Omron Sysmac Studio project 17-701_20171123 (Sysmac Studio 1.19.0.13, StandardProject)

# Controller new_Controller_0: NJ101-1000 version 1.13
Units and slaves: 電源 : NJ-Px3001; CPU : NJ101-1000; 0 : CJ1W-ID211 (J01); 1 : CJ1W-OD211 (J02)
Task PrimaryTask (priority 4, period or condition 2000): prIndexDataChange, prIndex, prStation1_PanelLoad, prStation1_FeedPanelLoad, prError, prStation1_PanelUnLoad, prStation1_FeedPanelUnLoad, prSystemInit, prStation1, prStation16, prStation4, prStation4_TH, prStation2

TYPE stIndexData : STRUCT
    FinishFlag : ARRAY[0..19] OF BOOL;
    OKFlag : ARRAY[0..19] OF BOOL;
    NGFlag : ARRAY[0..19] OF BOOL;
    ErrorLog : ARRAY[0..19] OF INT;
END_STRUCT END_TYPE

VAR_GLOBAL
    LS_S1_Load_PanelUpDown1Back : BOOL;  (* at ECAT://node#[1,1]/Input Bit 16 bits/Input Bit 00; published *)
    LS_S1_Load_PanelUpDown1Out : BOOL;  (* at ECAT://node#[1,1]/Input Bit 16 bits/Input Bit 01; published *)
    LS_S1_Load_PanelUpDown2Back : BOOL;  (* at ECAT://node#[1,1]/Input Bit 16 bits/Input Bit 02; published *)
    LS_S1_Load_PanelUpDown2Out : BOOL;  (* at ECAT://node#[1,1]/Input Bit 16 bits/Input Bit 03; published *)
    LS_S1_Load_PanelClip1Back : BOOL;  (* at ECAT://node#[1,1]/Input Bit 16 bits/Input Bit 04; published *)
    LS_S1_Load_PanelClip1Out : BOOL;  (* at ECAT://node#[1,1]/Input Bit 16 bits/Input Bit 05; published *)
    LS_S1_Load_PanelClip2Back : BOOL;  (* at ECAT://node#[1,1]/Input Bit 16 bits/Input Bit 06; published *)
    LS_S1_Load_PanelClip2Out : BOOL;  (* at ECAT://node#[1,1]/Input Bit 16 bits/Input Bit 07; published *)
    LS_S1_Load_FixClipBack : BOOL;  (* at ECAT://node#[1,1]/Input Bit 16 bits/Input Bit 08; published *)
    LS_S1_Load_FixClipOut : BOOL;  (* at ECAT://node#[1,1]/Input Bit 16 bits/Input Bit 09; published *)
    LS_S1_Load_AlignmentClipBack : BOOL;  (* at ECAT://node#[1,1]/Input Bit 16 bits/Input Bit 10; published *)
    LS_S1_Load_AlignmentClipOut : BOOL;  (* at ECAT://node#[1,1]/Input Bit 16 bits/Input Bit 11; published *)
    LS_S1_Load_ConveyorClip1Back : BOOL;  (* at ECAT://node#[1,1]/Input Bit 16 bits/Input Bit 12; published *)
    LS_S1_Load_ConveyorClip1Out : BOOL;  (* at ECAT://node#[1,1]/Input Bit 16 bits/Input Bit 13; published *)
    LS_S1_Load_ConveyorClip2Back : BOOL;  (* at ECAT://node#[1,1]/Input Bit 16 bits/Input Bit 14; published *)
    LS_S1_Load_ConveyorClip2Out : BOOL;  (* at ECAT://node#[1,1]/Input Bit 16 bits/Input Bit 15; published *)
    LS_S1_Load_UpDownBack : BOOL;  (* at ECAT://node#[1,2]/Input Bit 16 bits/Input Bit 00; published *)
    LS_S1_Load_UpDownOut : BOOL;  (* at ECAT://node#[1,2]/Input Bit 16 bits/Input Bit 01; published *)
    LS_S1_UnLoad_UpDownBack : BOOL;  (* at ECAT://node#[1,2]/Input Bit 16 bits/Input Bit 02; published *)
    LS_S1_UnLoad_UpDownOut : BOOL;  (* at ECAT://node#[1,2]/Input Bit 16 bits/Input Bit 03; published *)
    LS_S1_UnLoad_ConveyorClip1Back : BOOL;  (* at ECAT://node#[1,2]/Input Bit 16 bits/Input Bit 04; published *)
    LS_S1_UnLoad_ConveyorClip1Out : BOOL;  (* at ECAT://node#[1,2]/Input Bit 16 bits/Input Bit 05; published *)
    LS_S1_UnLoad_ConveyorClip2Back : BOOL;  (* at ECAT://node#[1,2]/Input Bit 16 bits/Input Bit 06; published *)
    LS_S1_UnLoad_ConveyorClip2Out : BOOL;  (* at ECAT://node#[1,2]/Input Bit 16 bits/Input Bit 07; published *)
    LS_S1_UnLoad_FixClipBack : BOOL;  (* at ECAT://node#[1,2]/Input Bit 16 bits/Input Bit 08; published *)
    LS_S1_UnLoad_FixClipOut : BOOL;  (* at ECAT://node#[1,2]/Input Bit 16 bits/Input Bit 09; published *)
    LS_S1_UnLoad_AlignmentClipBack : BOOL;  (* at ECAT://node#[1,2]/Input Bit 16 bits/Input Bit 10; published *)
    LS_S1_UnLoad_AlignmentClipOut : BOOL;  (* at ECAT://node#[1,2]/Input Bit 16 bits/Input Bit 11; published *)
    LS_S1_UnLoad_PanelClip1Back : BOOL;  (* at ECAT://node#[1,2]/Input Bit 16 bits/Input Bit 12; published *)
    LS_S1_UnLoad_PanelClip1Out : BOOL;  (* at ECAT://node#[1,2]/Input Bit 16 bits/Input Bit 13; published *)
    LS_S1_UnLoad_PanelClip2Back : BOOL;  (* at ECAT://node#[1,2]/Input Bit 16 bits/Input Bit 14; published *)
    LS_S1_UnLoad_PanelClip2Out : BOOL;  (* at ECAT://node#[1,2]/Input Bit 16 bits/Input Bit 15; published *)
    LS_S1_UnLoad_PanelUpDown1Back : BOOL;  (* at ECAT://node#[1,3]/Input Bit 16 bits/Input Bit 00; published *)
    LS_S1_UnLoad_PanelUpDown1Out : BOOL;  (* at ECAT://node#[1,3]/Input Bit 16 bits/Input Bit 01; published *)
    LS_S1_UnLoad_PanelUpDown2Back : BOOL;  (* at ECAT://node#[1,3]/Input Bit 16 bits/Input Bit 02; published *)
    LS_S1_UnLoad_PanelUpDown2Out : BOOL;  (* at ECAT://node#[1,3]/Input Bit 16 bits/Input Bit 03; published *)
    SNR_S1_Load_Full : BOOL;  (* 出盤缺盤檢知; at ECAT://node#[1,3]/Input Bit 16 bits/Input Bit 08; published *)
    SNR_S1_UnLoad_Full : BOOL;  (* 收盤滿盤檢知; at ECAT://node#[1,3]/Input Bit 16 bits/Input Bit 09; published *)
    SNR_S1_Load_Feed : BOOL;  (* 下移載出盤檢知; at ECAT://node#[1,3]/Input Bit 16 bits/Input Bit 10; published *)
    SNR_S1_UnLoad_Feed : BOOL;  (* 下移載收盤檢知; at ECAT://node#[1,3]/Input Bit 16 bits/Input Bit 11; published *)
    SNR_S1_Load_PanelFeed : BOOL;  (* 出盤下盤處檢知; at ECAT://node#[1,3]/Input Bit 16 bits/Input Bit 12; published *)
    SNR_S1_Load_PanelClip : BOOL;  (* 出盤夾盤處檢知; at ECAT://node#[1,3]/Input Bit 16 bits/Input Bit 13; published *)
    SNR_S1_UnLoad_PanelFeed : BOOL;  (* 收盤上盤處檢知; at ECAT://node#[1,3]/Input Bit 16 bits/Input Bit 14; published *)
    SNR_S1_UnLoad_PanelClip : BOOL;  (* 收盤夾盤處檢知; at ECAT://node#[1,3]/Input Bit 16 bits/Input Bit 15; published *)
    SOL_S1_Load_PanelUpDown1Back : BOOL;  (* at ECAT://node#[1,4]/Output Bit 16 bits/Output Bit 00; published *)
    SOL_S1_Load_PanelUpDown1Out : BOOL;  (* at ECAT://node#[1,4]/Output Bit 16 bits/Output Bit 01; published *)
    SOL_S1_Load_PanelUpDown2Back : BOOL;  (* at ECAT://node#[1,4]/Output Bit 16 bits/Output Bit 02; published *)
    SOL_S1_Load_PanelUpDown2Out : BOOL;  (* at ECAT://node#[1,4]/Output Bit 16 bits/Output Bit 03; published *)
    SOL_S1_Load_PanelClip : BOOL;  (* at ECAT://node#[1,4]/Output Bit 16 bits/Output Bit 04; published *)
    SOL_S1_Load_FixClip : BOOL;  (* at ECAT://node#[1,4]/Output Bit 16 bits/Output Bit 05; published *)
    SOL_S1_Load_AlignmentClip : BOOL;  (* at ECAT://node#[1,4]/Output Bit 16 bits/Output Bit 06; published *)
    SOL_S1_Load_ConveyorClip : BOOL;  (* at ECAT://node#[1,4]/Output Bit 16 bits/Output Bit 07; published *)
    SOL_S1_Load_UpDown : BOOL;  (* at ECAT://node#[1,4]/Output Bit 16 bits/Output Bit 08; published *)
    RY_S1_Load_FixSpeedMotor : BOOL;  (* at ECAT://node#[1,4]/Output Bit 16 bits/Output Bit 09; published *)
    RY_S1_UnLoad_FixSpeedMotor : BOOL;  (* at ECAT://node#[1,4]/Output Bit 16 bits/Output Bit 10; published *)
    RY_S1_Load_VariableSpeedMotor : BOOL;  (* at ECAT://node#[1,4]/Output Bit 16 bits/Output Bit 11; published *)
    RY_S1_UnLoad_VariableSpeedMotor : BOOL;  (* at ECAT://node#[1,4]/Output Bit 16 bits/Output Bit 12; published *)
    RY_S1_Center_VariableSpeedMotor : BOOL;  (* at ECAT://node#[1,4]/Output Bit 16 bits/Output Bit 13; published *)
    SOL_S1_UnLoad_PanelUpDown1Back : BOOL;  (* at ECAT://node#[1,8]/Output Bit 16 bits/Output Bit 00; published *)
    SOL_S1_UnLoad_PanelUpDown1Out : BOOL;  (* at ECAT://node#[1,8]/Output Bit 16 bits/Output Bit 01; published *)
    SOL_S1_UnLoad_PanelUpDown2Back : BOOL;  (* at ECAT://node#[1,8]/Output Bit 16 bits/Output Bit 02; published *)
    SOL_S1_UnLoad_PanelUpDown2Out : BOOL;  (* at ECAT://node#[1,8]/Output Bit 16 bits/Output Bit 03; published *)
    SOL_S1_UnLoad_PanelClip : BOOL;  (* at ECAT://node#[1,8]/Output Bit 16 bits/Output Bit 04; published *)
    SOL_S1_UnLoad_FixClip : BOOL;  (* at ECAT://node#[1,8]/Output Bit 16 bits/Output Bit 05; published *)
    SOL_S1_UnLoad_AlignmentClip : BOOL;  (* at ECAT://node#[1,8]/Output Bit 16 bits/Output Bit 06; published *)
    SOL_S1_UnLoad_ConveyorClip : BOOL;  (* at ECAT://node#[1,8]/Output Bit 16 bits/Output Bit 07; published *)
    SOL_S1_UnLoad_UpDown : BOOL;  (* at ECAT://node#[1,8]/Output Bit 16 bits/Output Bit 08; published *)
    YAMAHA_Unload_OKStart : BOOL;  (* at ECAT://node#[1,5]/Output Bit 16 bits/Output Bit 00; published *)
    YAMAHA_Unload_NGStart : BOOL;  (* at ECAT://node#[1,5]/Output Bit 16 bits/Output Bit 01; published *)
    YAMAHA_Load_Start : BOOL;  (* at ECAT://node#[1,5]/Output Bit 16 bits/Output Bit 02; published *)
    YAMAHA_UnLoad_Ready : BOOL;  (* at ECAT://node#[1,5]/Output Bit 16 bits/Output Bit 03; published *)
    YAMAHA_Load_Ready : BOOL;  (* at ECAT://node#[1,5]/Output Bit 16 bits/Output Bit 04; published *)
    YAMAHA_SOL_Clip : BOOL;  (* published *)
    YAMAHA_Error_SOL_Clip : BOOL;  (* at ECAT://node#[1,6]/Input Bit 16 bits/Input Bit 00; published *)
    YAMAHA_Unload_Finish : BOOL;  (* at ECAT://node#[1,6]/Input Bit 16 bits/Input Bit 01; published *)
    YAMAHA_Load_Finish : BOOL;  (* at ECAT://node#[1,6]/Input Bit 16 bits/Input Bit 02; published *)
    YAMAHA_Unload_ChangePanelStart : BOOL;  (* at ECAT://node#[1,6]/Input Bit 16 bits/Input Bit 03; published *)
    YAMAHA_Load_ChangePanelStart : BOOL;  (* at ECAT://node#[1,6]/Input Bit 16 bits/Input Bit 04; published *)
    YAMAHA_ORG : BOOL;  (* at ECAT://node#[1,6]/Input Bit 16 bits/Input Bit 05; published *)
    YAMAHA_S_Enable : BOOL;  (* at ECAT://node#[1,5]/Output Bit 16 bits/Output Bit 08; published *)
    YAMAHA_S_Control : BOOL;  (* at ECAT://node#[1,5]/Output Bit 16 bits/Output Bit 09; published *)
    YAMAHA_S_Stop : BOOL;  (* at ECAT://node#[1,5]/Output Bit 16 bits/Output Bit 10; published *)
    YAMAHA_S_AutoRun : BOOL;  (* at ECAT://node#[1,5]/Output Bit 16 bits/Output Bit 11; published *)
    YAMAHA_S_INCHome : BOOL;  (* at ECAT://node#[1,5]/Output Bit 16 bits/Output Bit 12; published *)
    YAMAHA_S_ProgramReset : BOOL;  (* at ECAT://node#[1,5]/Output Bit 16 bits/Output Bit 13; published *)
    YAMAHA_S_AlarmReset : BOOL;  (* at ECAT://node#[1,5]/Output Bit 16 bits/Output Bit 14; published *)
    YAMAHA_S_ABSHome : BOOL;  (* at ECAT://node#[1,5]/Output Bit 16 bits/Output Bit 15; published *)
    YAMAHA_S_State_CPUOK : BOOL;  (* at ECAT://node#[1,6]/Input Bit 16 bits/Input Bit 08; published *)
    YAMAHA_S_State_AutoMode : BOOL;  (* at ECAT://node#[1,6]/Input Bit 16 bits/Input Bit 09; published *)
    YAMAHA_S_State_Homed : BOOL;  (* at ECAT://node#[1,6]/Input Bit 16 bits/Input Bit 10; published *)
    YAMAHA_S_State_RobotProgramRun : BOOL;  (* at ECAT://node#[1,6]/Input Bit 16 bits/Input Bit 11; published *)
    YAMAHA_S_State_ProgramReset : BOOL;  (* at ECAT://node#[1,6]/Input Bit 16 bits/Input Bit 12; published *)
    YAMAHA_S_State_Warring : BOOL;  (* at ECAT://node#[1,6]/Input Bit 16 bits/Input Bit 13; published *)
    YAMAHA_S_State_Enable : BOOL;  (* at ECAT://node#[1,6]/Input Bit 16 bits/Input Bit 14; published *)
    YAMAHA_S_State_Alarm : BOOL;  (* at ECAT://node#[1,6]/Input Bit 16 bits/Input Bit 15; published *)
    SNR_S1_Door1 : BOOL;  (* at ECAT://node#[1,3]/Input Bit 16 bits/Input Bit 04; published *)
    SNR_S1_Door2 : BOOL;  (* at ECAT://node#[1,3]/Input Bit 16 bits/Input Bit 05; published *)
    SNR_S1_Door3 : BOOL;  (* at ECAT://node#[1,3]/Input Bit 16 bits/Input Bit 06; published *)
    SNR_S1_Door4 : BOOL;  (* at ECAT://node#[1,3]/Input Bit 16 bits/Input Bit 07; published *)
    LS_S4_Load_PanelUpDown1Back : BOOL;  (* published *)
    LS_S4_Load_PanelUpDown1Out : BOOL;  (* published *)
    LS_S4_Load_PanelUpDown2Back : BOOL;  (* published *)
    LS_S4_Load_PanelUpDown2Out : BOOL;  (* published *)
    LS_S4_Load_PanelClip1Back : BOOL;  (* published *)
    LS_S4_Load_PanelClip1Out : BOOL;  (* published *)
    LS_S4_Load_PanelClip2Back : BOOL;  (* published *)
    LS_S4_Load_PanelClip2Out : BOOL;  (* published *)
    LS_S4_UnLoad_PanelUpDown1Back : BOOL;  (* published *)
    LS_S4_UnLoad_PanelUpDown1Out : BOOL;  (* published *)
    LS_S4_UnLoad_PanelUpDown2Back : BOOL;  (* published *)
    LS_S4_UnLoad_PanelUpDown2Out : BOOL;  (* published *)
    LS_S4_UnLoad_PanelClip1Back : BOOL;  (* published *)
    LS_S4_UnLoad_PanelClip1Out : BOOL;  (* published *)
    LS_S4_UnLoad_PanelClip2Back : BOOL;  (* published *)
    LS_S4_UnLoad_PanelClip2Out : BOOL;  (* published *)
    LS_S4_Center_UpDownBack : BOOL;  (* published *)
    LS_S4_Center_UpDownOut : BOOL;  (* published *)
    LS_S4_Center_ClipBack : BOOL;  (* published *)
    LS_S4_Center_ClipOut : BOOL;  (* published *)
    SNR_S4_Load_Feed : BOOL;  (* published *)
    SNR_S4_UnLoad_Feed : BOOL;  (* published *)
    SNR_S4_Load_Full : BOOL;  (* published *)
    SNR_S4_UnLoad_Full : BOOL;  (* published *)
    SOL_S4_Load_PanelUpDown1Back : BOOL;  (* published *)
    SOL_S4_Load_PanelUpDown1Out : BOOL;  (* published *)
    SOL_S4_Load_PanelUpDown2Back : BOOL;  (* published *)
    SOL_S4_Load_PanelUpDown2Out : BOOL;  (* published *)
    SOL_S4_Load_PanelClip : BOOL;  (* published *)
    SOL_S4_UnLoad_PanelUpDown1Back : BOOL;  (* published *)
    SOL_S4_UnLoad_PanelUpDown1Out : BOOL;  (* published *)
    SOL_S4_UnLoad_PanelUpDown2Back : BOOL;  (* published *)
    SOL_S4_UnLoad_PanelUpDown2Out : BOOL;  (* published *)
    SOL_S4_UnLoad_PanelClip : BOOL;  (* published *)
    SOL_S4_Center_UpDown : BOOL;  (* published *)
    SOL_S4_Center_Clip : BOOL;  (* published *)
    SOL_S2_UpDown : BOOL;  (* published *)
    SOL_S4_MoveBack : BOOL;  (* published *)
    SOL_S4_MoveOut : BOOL;  (* published *)
    SOL_S4_UpDown : BOOL;  (* published *)
    SOL_S4_Clip : BOOL;  (* published *)
    SOL_S4_THMoveBack : BOOL;  (* published *)
    SOL_S4_THMoveOut : BOOL;  (* published *)
    SOL_S6_MoveBack : BOOL;  (* published *)
    SOL_S6_MoveOut : BOOL;  (* published *)
    SOL_S6_UpDown : BOOL;  (* published *)
    SOL_S6_TH : BOOL;  (* published *)
    SOL_S8_MoveBack : BOOL;  (* published *)
    SOL_S8_MoveOut : BOOL;  (* published *)
    SOL_S8_UpDown : BOOL;  (* published *)
    SOL_S8_FixMove : BOOL;  (* published *)
    SOL_S8_Fix : BOOL;  (* published *)
    SOL_S8_TH : BOOL;  (* published *)
    SOL_S8_Turn : BOOL;  (* published *)
    SOL_S8_Clip : BOOL;  (* published *)
    SOL_S10_MoveBack : BOOL;  (* published *)
    SOL_S10_MoveOut : BOOL;  (* published *)
    SOL_S10_UpDown : BOOL;  (* published *)
    SOL_S10_ClipF : BOOL;  (* published *)
    SOL_S10_ClipR : BOOL;  (* published *)
    SOL_S10_TH : BOOL;  (* published *)
    SOL_S10_Turn : BOOL;  (* published *)
    SOL_S11_UpDown : BOOL;  (* published *)
    SOL_S13_UpDown : BOOL;  (* published *)
    SOL_S15_UpDown : BOOL;  (* published *)
    SOL_S6_Vacuum : BOOL;  (* published *)
    SOL_S6_Break : BOOL;  (* published *)
    SOL_S8_VacuumF : BOOL;  (* published *)
    SOL_S8_BreakF : BOOL;  (* published *)
    SOL_S8_VacuumR : BOOL;  (* published *)
    SOL_S8_BreakR : BOOL;  (* published *)
    RY_S6_Full : BOOL;  (* published *)
    RY_S6_Feed : BOOL;  (* published *)
    RY_S8_Full : BOOL;  (* published *)
    RY_S8_Feed : BOOL;  (* published *)
    RY_S10_Full : BOOL;  (* published *)
    RY_S10_Feed : BOOL;  (* published *)
    LS_S2_UpDownBack : BOOL;  (* published *)
    LS_S2_UpDownOut : BOOL;  (* published *)
    LS_S4_MoveBack : BOOL;  (* published *)
    LS_S4_MoveOut : BOOL;  (* published *)
    LS_S4_UpDownBack : BOOL;  (* published *)
    LS_S4_UpDownOut : BOOL;  (* published *)
    LS_S4_ClipBack : BOOL;  (* published *)
    LS_S4_ClipOut : BOOL;  (* published *)
    LS_S4_THMoveBack : BOOL;  (* published *)
    LS_S4_THMoveOut : BOOL;  (* published *)
    LS_S6_MoveBack : BOOL;  (* published *)
    LS_S6_MoveOut : BOOL;  (* published *)
    LS_S6_UpDownBack : BOOL;  (* published *)
    LS_S6_UpDownOut : BOOL;  (* published *)
    LS_S6_THBack : BOOL;  (* published *)
    LS_S6_THOut : BOOL;  (* published *)
    LS_S8_MoveBack : BOOL;  (* published *)
    LS_S8_MoveOut : BOOL;  (* published *)
    LS_S8_UpDownBack : BOOL;  (* published *)
    LS_S8_UpDownOut : BOOL;  (* published *)
    LS_S8_FixMoveBack : BOOL;  (* published *)
    LS_S8_FixMoveOut : BOOL;  (* published *)
    LS_S8_FixBack : BOOL;  (* published *)
    LS_S8_FixOut : BOOL;  (* published *)
    LS_S8_THBack : BOOL;  (* published *)
    LS_S8_THOut : BOOL;  (* published *)
    LS_S8_TurnBack : BOOL;  (* published *)
    LS_S8_TurnOut : BOOL;  (* published *)
    LS_S8_ClipBack : BOOL;  (* published *)
    LS_S8_ClipOut : BOOL;  (* published *)
    LS_S10_MoveBack : BOOL;  (* published *)
    LS_S10_MoveOut : BOOL;  (* published *)
    LS_S10_UpDownBack : BOOL;  (* published *)
    LS_S10_UpDownOut : BOOL;  (* published *)
    LS_S10_ClipFBack : BOOL;  (* published *)
    LS_S10_ClipFOut : BOOL;  (* published *)
    LS_S10_ClipRBack : BOOL;  (* published *)
    LS_S10_ClipROut : BOOL;  (* published *)
    LS_S10_THBack : BOOL;  (* published *)
    LS_S10_THOut : BOOL;  (* published *)
    LS_S10_TurnBack : BOOL;  (* published *)
    LS_S10_TurnOut : BOOL;  (* published *)
    LS_S11_UpDownBack : BOOL;  (* published *)
    LS_S11_UpDownOut : BOOL;  (* published *)
    LS_S13_UpDownBack : BOOL;  (* published *)
    LS_S13_UpDownOut : BOOL;  (* published *)
    LS_S15_UpDownBack : BOOL;  (* published *)
    LS_S15_UpDownOut : BOOL;  (* published *)
    LS_S13_TempHighWarring : BOOL;  (* published *)
    LS_S13_TempLowWarring : BOOL;  (* published *)
    SNR_S4_Feed : BOOL;  (* published *)
    SNR_S5_Check : BOOL;  (* published *)
    SNR_S6_Vacuum : BOOL;  (* published *)
    SNR_S6_Full : BOOL;  (* published *)
    SNR_S6_Feed : BOOL;  (* published *)
    SNR_S7_Check : BOOL;  (* published *)
    SNR_S8_VacuumF : BOOL;  (* published *)
    SNR_S8_VacuumR : BOOL;  (* published *)
    SNR_S8_Full : BOOL;  (* published *)
    SNR_S8_Feed : BOOL;  (* published *)
    SNR_S9_Check : BOOL;  (* published *)
    SNR_S10_Full : BOOL;  (* published *)
    SNR_S10_Feed : BOOL;  (* published *)
    SNR_Index : BOOL;  (* published *)
    SNR_AirSource : BOOL;  (* published *)
    OMRON_FQ2_NG : BOOL;  (* published *)
    OMRON_FQ2_Ready : BOOL;  (* published *)
    OMRON_FQ2_Error : BOOL;  (* published *)
    OMRON_FQ2_Trig : BOOL;  (* published *)
    OMRON_FQ2_IN0 : BOOL;  (* published *)
    OMRON_FQ2_IN1 : BOOL;  (* published *)
    OMRON_FQ2_IN2 : BOOL;  (* published *)
    OMRON_FQ2_IN3 : BOOL;  (* published *)
    OMRON_FQ2_IN4 : BOOL;  (* published *)
    OMRON_FQ2_IN5 : BOOL;  (* published *)
    RY_Index : BOOL;  (* published *)
    BZ : BOOL;  (* published *)
    YL : BOOL;  (* published *)
    GL : BOOL;  (* published *)
    RL : BOOL;  (* published *)
    Invertor_Ready : BOOL;  (* published *)
    PB_Start : BOOL;  (* published *)
    PB_Reset : BOOL;  (* published *)
    PB_EStop : BOOL;  (* published *)
    HMIPB_SOL_S1_Load_PanelUpDown1Back : BOOL;  (* published *)
    HMIPB_SOL_S1_Load_PanelUpDown1Out : BOOL;  (* published *)
    HMIPB_SOL_S1_Load_PanelUpDown2Back : BOOL;  (* published *)
    HMIPB_SOL_S1_Load_PanelUpDown2Out : BOOL;  (* published *)
    HMIPB_SOL_S1_Load_PanelClip : BOOL;  (* published *)
    HMIPB_SOL_S1_Load_FixClip : BOOL;  (* published *)
    HMIPB_SOL_S1_Load_AlignmentClip : BOOL;  (* published *)
    HMIPB_SOL_S1_Load_ConveyorClip : BOOL;  (* published *)
    HMIPB_SOL_S1_Load_UpDown : BOOL;  (* published *)
    HMIPB_RY_S1_Load_FixSpeedMotor : BOOL;  (* published *)
    HMIPB_RY_S1_UnLoad_FixSpeedMotor : BOOL;  (* published *)
    HMIPB_RY_S1_Load_VariableSpeedMotor : BOOL;  (* published *)
    HMIPB_RY_S1_UnLoad_VariableSpeedMotor : BOOL;  (* published *)
    HMIPB_RY_S1_Center_VariableSpeedMotor : BOOL;  (* published *)
    HMIPB_SOL_S1_UnLoad_PanelUpDown1Back : BOOL;  (* published *)
    HMIPB_SOL_S1_UnLoad_PanelUpDown1Out : BOOL;  (* published *)
    HMIPB_SOL_S1_UnLoad_PanelUpDown2Back : BOOL;  (* published *)
    HMIPB_SOL_S1_UnLoad_PanelUpDown2Out : BOOL;  (* published *)
    HMIPB_SOL_S1_UnLoad_PanelClip : BOOL;  (* published *)
    HMIPB_SOL_S1_UnLoad_FixClip : BOOL;  (* published *)
    HMIPB_SOL_S1_UnLoad_AlignmentClip : BOOL;  (* published *)
    HMIPB_SOL_S1_UnLoad_ConveyorClip : BOOL;  (* published *)
    HMIPB_SOL_S1_UnLoad_UpDown : BOOL;  (* published *)
    HMIPB_YAMAHA_Unload_OKStart : BOOL;  (* published *)
    HMIPB_YAMAHA_Unload_NGStart : BOOL;  (* published *)
    HMIPB_YAMAHA_Load_Start : BOOL;  (* published *)
    HMIPB_YAMAHA_UnLoad_Ready : BOOL;  (* published *)
    HMIPB_YAMAHA_Load_Ready : BOOL;  (* published *)
    HMIPB_YAMAHA_SOL_Clip : BOOL;  (* published *)
    HMIPB_YAMAHA_Unload_ChangePanelStart : BOOL;  (* published *)
    HMIPB_YAMAHA_Load_ChangePanelStart : BOOL;  (* published *)
    HMIPB_YAMAHA_ORG : BOOL;  (* published *)
    HMIPB_YAMAHA_S_Enable : BOOL;  (* published *)
    HMIPB_YAMAHA_S_Control : BOOL;  (* published *)
    HMIPB_YAMAHA_S_Stop : BOOL;  (* published *)
    HMIPB_YAMAHA_S_AutoRun : BOOL;  (* published *)
    HMIPB_YAMAHA_S_INCHome : BOOL;  (* published *)
    HMIPB_YAMAHA_S_ProgramReset : BOOL;  (* published *)
    HMIPB_YAMAHA_S_AlarmReset : BOOL;  (* published *)
    HMIPB_YAMAHA_S_ABSHome : BOOL;  (* published *)
    HMIPB_SOL_S4_Load_PanelUpDown1Back : BOOL;  (* published *)
    HMIPB_SOL_S4_Load_PanelUpDown1Out : BOOL;  (* published *)
    HMIPB_SOL_S4_Load_PanelUpDown2Back : BOOL;  (* published *)
    HMIPB_SOL_S4_Load_PanelUpDown2Out : BOOL;  (* published *)
    HMIPB_SOL_S4_Load_PanelClip : BOOL;  (* published *)
    HMIPB_SOL_S4_UnLoad_PanelUpDown1Back : BOOL;  (* published *)
    HMIPB_SOL_S4_UnLoad_PanelUpDown1Out : BOOL;  (* published *)
    HMIPB_SOL_S4_UnLoad_PanelUpDown2Back : BOOL;  (* published *)
    HMIPB_SOL_S4_UnLoad_PanelUpDown2Out : BOOL;  (* published *)
    HMIPB_SOL_S4_UnLoad_PanelClip : BOOL;  (* published *)
    HMIPB_SOL_S4_Center_UpDown : BOOL;  (* published *)
    HMIPB_SOL_S4_Center_Clip : BOOL;  (* published *)
    HMIPB_SOL_S2_UpDown : BOOL;  (* published *)
    HMIPB_SOL_S4_MoveBack : BOOL;  (* published *)
    HMIPB_SOL_S4_MoveOut : BOOL;  (* published *)
    HMIPB_SOL_S4_UpDown : BOOL;  (* published *)
    HMIPB_SOL_S4_Clip : BOOL;  (* published *)
    HMIPB_SOL_S4_THMoveBack : BOOL;  (* published *)
    HMIPB_SOL_S4_THMoveOut : BOOL;  (* published *)
    HMIPB_SOL_S6_MoveBack : BOOL;  (* published *)
    HMIPB_SOL_S6_MoveOut : BOOL;  (* published *)
    HMIPB_SOL_S6_UpDown : BOOL;  (* published *)
    HMIPB_SOL_S6_TH : BOOL;  (* published *)
    HMIPB_SOL_S8_MoveBack : BOOL;  (* published *)
    HMIPB_SOL_S8_MoveOut : BOOL;  (* published *)
    HMIPB_SOL_S8_UpDown : BOOL;  (* published *)
    HMIPB_SOL_S8_FixMove : BOOL;  (* published *)
    HMIPB_SOL_S8_Fix : BOOL;  (* published *)
    HMIPB_SOL_S8_TH : BOOL;  (* published *)
    HMIPB_SOL_S8_Turn : BOOL;  (* published *)
    HMIPB_SOL_S8_Clip : BOOL;  (* published *)
    HMIPB_SOL_S10_MoveBack : BOOL;  (* published *)
    HMIPB_SOL_S10_MoveOut : BOOL;  (* published *)
    HMIPB_SOL_S10_UpDown : BOOL;  (* published *)
    HMIPB_SOL_S10_ClipF : BOOL;  (* published *)
    HMIPB_SOL_S10_ClipR : BOOL;  (* published *)
    HMIPB_SOL_S10_TH : BOOL;  (* published *)
    HMIPB_SOL_S10_Turn : BOOL;  (* published *)
    HMIPB_SOL_S11_UpDown : BOOL;  (* published *)
    HMIPB_SOL_S13_UpDown : BOOL;  (* published *)
    HMIPB_SOL_S15_UpDown : BOOL;  (* published *)
    HMIPB_SOL_S6_Vacuum : BOOL;  (* published *)
    HMIPB_SOL_S6_Break : BOOL;  (* published *)
    HMIPB_SOL_S8_VacuumF : BOOL;  (* published *)
    HMIPB_SOL_S8_BreakF : BOOL;  (* published *)
    HMIPB_SOL_S8_VacuumR : BOOL;  (* published *)
    HMIPB_SOL_S8_BreakR : BOOL;  (* published *)
    HMIPB_RY_S6_Full : BOOL;  (* published *)
    HMIPB_RY_S6_Feed : BOOL;  (* published *)
    HMIPB_RY_S8_Full : BOOL;  (* published *)
    HMIPB_RY_S8_Feed : BOOL;  (* published *)
    HMIPB_RY_S10_Full : BOOL;  (* published *)
    HMIPB_RY_S10_Feed : BOOL;  (* published *)
    HMIPB_OMRON_FQ2_Trig : BOOL;  (* published *)
    HMIPB_RY_Index : BOOL;  (* published *)
    DisablePB : ARRAY[0..19] OF BOOL;  (* published *)
    TestPB : ARRAY[0..19] OF BOOL;  (* published *)
    Error_LS_S1_Load_PanelUpDown1Back : BOOL;  (* published *)
    Error_LS_S1_Load_PanelUpDown1Out : BOOL;  (* published *)
    Error_LS_S1_Load_PanelUpDown2Back : BOOL;  (* published *)
    Error_LS_S1_Load_PanelUpDown2Out : BOOL;  (* published *)
    Error_LS_S1_Load_PanelClip1Back : BOOL;  (* published *)
    Error_LS_S1_Load_PanelClip1Out : BOOL;  (* published *)
    Error_LS_S1_Load_PanelClip2Back : BOOL;  (* published *)
    Error_LS_S1_Load_PanelClip2Out : BOOL;  (* published *)
    Error_LS_S1_Load_FixClipBack : BOOL;  (* published *)
    Error_LS_S1_Load_FixClipOut : BOOL;  (* published *)
    Error_LS_S1_Load_AlignmentClipBack : BOOL;  (* published *)
    Error_LS_S1_Load_AlignmentClipOut : BOOL;  (* published *)
    Error_LS_S1_Load_ConveyorClip1Back : BOOL;  (* published *)
    Error_LS_S1_Load_ConveyorClip1Out : BOOL;  (* published *)
    Error_LS_S1_Load_ConveyorClip2Back : BOOL;  (* published *)
    Error_LS_S1_Load_ConveyorClip2Out : BOOL;  (* published *)
    Error_LS_S1_Load_UpDownBack : BOOL;  (* published *)
    Error_LS_S1_Load_UpDownOut : BOOL;  (* published *)
    Error_LS_S1_UnLoad_UpDownBack : BOOL;  (* published *)
    Error_LS_S1_UnLoad_UpDownOut : BOOL;  (* published *)
    Error_LS_S1_UnLoad_ConveyorClip1Back : BOOL;  (* published *)
    Error_LS_S1_UnLoad_ConveyorClip1Out : BOOL;  (* published *)
    Error_LS_S1_UnLoad_ConveyorClip2Back : BOOL;  (* published *)
    Error_LS_S1_UnLoad_ConveyorClip2Out : BOOL;  (* published *)
    Error_LS_S1_UnLoad_FixClipBack : BOOL;  (* published *)
    Error_LS_S1_UnLoad_FixClipOut : BOOL;  (* published *)
    Error_LS_S1_UnLoad_AlignmentClipBack : BOOL;  (* published *)
    Error_LS_S1_UnLoad_AlignmentClipOut : BOOL;  (* published *)
    Error_LS_S1_UnLoad_PanelClip1Back : BOOL;  (* published *)
    Error_LS_S1_UnLoad_PanelClip1Out : BOOL;  (* published *)
    Error_LS_S1_UnLoad_PanelClip2Back : BOOL;  (* published *)
    Error_LS_S1_UnLoad_PanelClip2Out : BOOL;  (* published *)
    Error_LS_S1_UnLoad_PanelUpDown1Back : BOOL;  (* published *)
    Error_LS_S1_UnLoad_PanelUpDown1Out : BOOL;  (* published *)
    Error_LS_S1_UnLoad_PanelUpDown2Back : BOOL;  (* published *)
    Error_LS_S1_UnLoad_PanelUpDown2Out : BOOL;  (* published *)
    Error_SNR_S1_Load_Full : BOOL;  (* published *)
    Error_SNR_S1_UnLoad_Full : BOOL;  (* published *)
    Error_SNR_S1_Load_Feed : BOOL;  (* published *)
    Error_SNR_S1_UnLoad_Feed : BOOL;  (* published *)
    Error_SNR_S1_Load_PanelFeed : BOOL;  (* published *)
    Error_SNR_S1_Load_PanelClip : BOOL;  (* published *)
    Error_SNR_S1_UnLoad_PanelFeed : BOOL;  (* published *)
    Error_SNR_S1_UnLoad_PanelClip : BOOL;  (* published *)
    Error_YAMAHA_Error_SOL_Clip : BOOL;  (* published *)
    Error_YAMAHA_S_State_Warring : BOOL;  (* published *)
    Error_YAMAHA_S_State_Alarm : BOOL;  (* published *)
    Error_LS_S4_Load_PanelUpDown1Back : BOOL;  (* published *)
    Error_LS_S4_Load_PanelUpDown1Out : BOOL;  (* published *)
    Error_LS_S4_Load_PanelUpDown2Back : BOOL;  (* published *)
    Error_LS_S4_Load_PanelUpDown2Out : BOOL;  (* published *)
    Error_LS_S4_Load_PanelClip1Back : BOOL;  (* published *)
    Error_LS_S4_Load_PanelClip1Out : BOOL;  (* published *)
    Error_LS_S4_Load_PanelClip2Back : BOOL;  (* published *)
    Error_LS_S4_Load_PanelClip2Out : BOOL;  (* published *)
    Error_LS_S4_UnLoad_PanelUpDown1Back : BOOL;  (* published *)
    Error_LS_S4_UnLoad_PanelUpDown1Out : BOOL;  (* published *)
    Error_LS_S4_UnLoad_PanelUpDown2Back : BOOL;  (* published *)
    Error_LS_S4_UnLoad_PanelUpDown2Out : BOOL;  (* published *)
    Error_LS_S4_UnLoad_PanelClip1Back : BOOL;  (* published *)
    Error_LS_S4_UnLoad_PanelClip1Out : BOOL;  (* published *)
    Error_LS_S4_UnLoad_PanelClip2Back : BOOL;  (* published *)
    Error_LS_S4_UnLoad_PanelClip2Out : BOOL;  (* published *)
    Error_LS_S4_Center_UpDownBack : BOOL;  (* published *)
    Error_LS_S4_Center_UpDownOut : BOOL;  (* published *)
    Error_LS_S4_Center_ClipBack : BOOL;  (* published *)
    Error_LS_S4_Center_ClipOut : BOOL;  (* published *)
    Error_SNR_S4_Load_Feed : BOOL;  (* published *)
    Error_SNR_S4_UnLoad_Feed : BOOL;  (* published *)
    Error_SNR_S4_Load_Full : BOOL;  (* published *)
    Error_SNR_S4_UnLoad_Full : BOOL;  (* published *)
    Error_LS_S2_UpDownBack : BOOL;  (* published *)
    Error_LS_S2_UpDownOut : BOOL;  (* published *)
    Error_LS_S4_MoveBack : BOOL;  (* published *)
    Error_LS_S4_MoveOut : BOOL;  (* published *)
    Error_LS_S4_UpDownBack : BOOL;  (* published *)
    Error_LS_S4_UpDownOut : BOOL;  (* published *)
    Error_LS_S4_ClipBack : BOOL;  (* published *)
    Error_LS_S4_ClipOut : BOOL;  (* published *)
    Error_LS_S4_THMoveBack : BOOL;  (* published *)
    Error_LS_S4_THMoveOut : BOOL;  (* published *)
    Error_LS_S6_MoveBack : BOOL;  (* published *)
    Error_LS_S6_MoveOut : BOOL;  (* published *)
    Error_LS_S6_UpDownBack : BOOL;  (* published *)
    Error_LS_S6_UpDownOut : BOOL;  (* published *)
    Error_LS_S6_THBack : BOOL;  (* published *)
    Error_LS_S6_THOut : BOOL;  (* published *)
    Error_LS_S8_MoveBack : BOOL;  (* published *)
    Error_LS_S8_MoveOut : BOOL;  (* published *)
    Error_LS_S8_UpDownBack : BOOL;  (* published *)
    Error_LS_S8_UpDownOut : BOOL;  (* published *)
    Error_LS_S8_FixMoveBack : BOOL;  (* published *)
    Error_LS_S8_FixMoveOut : BOOL;  (* published *)
    Error_LS_S8_FixBack : BOOL;  (* published *)
    Error_LS_S8_FixOut : BOOL;  (* published *)
    Error_LS_S8_THBack : BOOL;  (* published *)
    Error_LS_S8_THOut : BOOL;  (* published *)
    Error_LS_S8_TurnBack : BOOL;  (* published *)
    Error_LS_S8_TurnOut : BOOL;  (* published *)
    Error_LS_S8_ClipBack : BOOL;  (* published *)
    Error_LS_S8_ClipOut : BOOL;  (* published *)
    Error_LS_S10_MoveBack : BOOL;  (* published *)
    Error_LS_S10_MoveOut : BOOL;  (* published *)
    Error_LS_S10_UpDownBack : BOOL;  (* published *)
    Error_LS_S10_UpDownOut : BOOL;  (* published *)
    Error_LS_S10_ClipFBack : BOOL;  (* published *)
    Error_LS_S10_ClipFOut : BOOL;  (* published *)
    Error_LS_S10_ClipRBack : BOOL;  (* published *)
    Error_LS_S10_ClipROut : BOOL;  (* published *)
    Error_LS_S10_THBack : BOOL;  (* published *)
    Error_LS_S10_THOut : BOOL;  (* published *)
    Error_LS_S10_TurnBack : BOOL;  (* published *)
    Error_LS_S10_TurnOut : BOOL;  (* published *)
    Error_LS_S11_UpDownBack : BOOL;  (* published *)
    Error_LS_S11_UpDownOut : BOOL;  (* published *)
    Error_LS_S13_UpDownBack : BOOL;  (* published *)
    Error_LS_S13_UpDownOut : BOOL;  (* published *)
    Error_LS_S15_UpDownBack : BOOL;  (* published *)
    Error_LS_S15_UpDownOut : BOOL;  (* published *)
    Error_LS_S13_TempHighWarring : BOOL;  (* published *)
    Error_LS_S13_TempLowWarring : BOOL;  (* published *)
    Error_SNR_S4_Feed : BOOL;  (* published *)
    Error_SNR_S5_Check : BOOL;  (* published *)
    Error_SNR_S6_Vacuum : BOOL;  (* published *)
    Error_SNR_S6_Full : BOOL;  (* published *)
    Error_SNR_S6_Feed : BOOL;  (* published *)
    Error_SNR_S7_Check : BOOL;  (* published *)
    Error_SNR_S8_VacuumF : BOOL;  (* published *)
    Error_SNR_S8_VacuumR : BOOL;  (* published *)
    Error_SNR_S8_Full : BOOL;  (* published *)
    Error_SNR_S8_Feed : BOOL;  (* published *)
    Error_SNR_S9_Check : BOOL;  (* published *)
    Error_SNR_S10_Full : BOOL;  (* published *)
    Error_SNR_S10_Feed : BOOL;  (* published *)
    Error_SNR_Index : BOOL;  (* published *)
    Error_SNR_AirSource : BOOL;  (* published *)
    Error_OMRON_FQ2_Error : BOOL;  (* published *)
    Error_Invertor_Ready : BOOL;  (* published *)
    Error_PB_EStop : BOOL;  (* published *)
    AutoStatus : BOOL;  (* published *)
    SystemReadyStatus : BOOL;
    MachineRunStatus : BOOL;
    Manual2AutoFlag : BOOL;
    FeedStart : ARRAY[0..19] OF BOOL;
    FeedFinish : ARRAY[0..19] OF BOOL;
    ErrorStatus : ARRAY[0..19] OF BOOL;
    ErrorStatus_TH : ARRAY[0..19] OF BOOL;
    ErrorStatus_S1_Load : BOOL;
    ErrorStatus_S1_FeedPanelLoad : BOOL;
    ErrorStatus_S1_UnLoad : BOOL;
    ErrorStatus_S1_FeedPanelUnLoad : BOOL;
    ErrorStatus_S1_Center : BOOL;
    ErrorStatus_S4_Load : BOOL;
    ErrorStatus_S4_UnLoad : BOOL;
    ErrorStatus_S4_Center : BOOL;
    ErrorStatus_MachineStop : BOOL;
    ErrorStatus_MachineStop_Record : BOOL;
    ErrorStatus_MachineNonStop : BOOL;
END_VAR
VAR_GLOBAL RETAIN
    IndexData : ARRAY[0..19] OF stIndexData;  (* published *)
    TotalCount : DINT;  (* published *)
    OKCount : DINT;  (* published *)
    NGCount : DINT;  (* published *)
    HMISV_Index_DelayTime : DINT;  (* published *)
END_VAR

PROGRAM prIndexDataChange
VAR
    R_TRIG_1 : R_TRIG;
END_VAR
VAR_EXTERNAL
    SNR_Index : BOOL;
    IndexData : array[0..19] of stIndexData;
    OKCount : DINT;
    NGCount : DINT;
    SystemReadyStatus : BOOL;
END_VAR
(*本機轉盤*)
R_TRIG_1(CLK:=SNR_Index);
IF SystemReadyStatus AND R_TRIG_1.Q THEN
	IndexData[19]:=IndexData[18];
	IndexData[18]:=IndexData[17];
	IndexData[17]:=IndexData[16];
	IndexData[16]:=IndexData[15];
	IndexData[15]:=IndexData[14];
	IndexData[14]:=IndexData[13];
	IndexData[13]:=IndexData[12];
	IndexData[12]:=IndexData[11];
	IndexData[11]:=IndexData[10];
	IndexData[10]:=IndexData[9];
	IndexData[9]:=IndexData[8];
	IndexData[8]:=IndexData[7];
	IndexData[7]:=IndexData[6];
	IndexData[6]:=IndexData[5];
	IndexData[5]:=IndexData[4];
	IndexData[4]:=IndexData[3];
	IndexData[3]:=IndexData[2];
	IndexData[2]:=IndexData[1];
	IndexData[1]:=IndexData[0];
END_IF;
(*計數器*)
IF SystemReadyStatus AND R_TRIG_1.Q THEN
	IF IndexData[16].OKFlag[2] AND IndexData[16].OKFlag[15] THEN
		OKCount:=OKCount+1;
	END_IF;
	IF IndexData[16].OKFlag[2] AND IndexData[16].OKFlag[15] THEN
		NGCount:=NGCount+1;
	END_IF;
END_IF;
END_PROGRAM

PROGRAM prIndex
VAR
    R_TRIG_1 : R_TRIG;
    tDelayTime : TIME;
    TON_1 : TON;
    IndexCanRunStatus : BOOL;
    Autoflow : INT;
END_VAR
VAR_EXTERNAL
    SystemReadyStatus : BOOL;
    HMIPB_RY_Index : BOOL;
    HMISV_Index_DelayTime : DINT;
    YAMAHA_ORG : BOOL;
    LS_S2_UpDownBack : BOOL;
    SOL_S2_UpDown : BOOL;
    LS_S4_UpDownBack : BOOL;
    RY_Index : BOOL;
    ErrorStatus : ARRAY[0..19] OF BOOL;
    AutoStatus : BOOL;
    MachineRunStatus : BOOL;
    IndexData : ARRAY[0..19] OF stIndexData;
    SNR_Index : BOOL;
    SOL_S4_UpDown : BOOL;
    LS_S4_MoveBack : BOOL;
    LS_S6_UpDownBack : BOOL;
    SOL_S6_UpDown : BOOL;
    LS_S6_MoveBack : BOOL;
    LS_S8_UpDownBack : BOOL;
    SOL_S8_UpDown : BOOL;
    LS_S8_MoveOut : BOOL;
    LS_S10_UpDownBack : BOOL;
    SOL_S10_UpDown : BOOL;
    LS_S10_MoveOut : BOOL;
    LS_S11_UpDownBack : BOOL;
    SOL_S11_UpDown : BOOL;
    LS_S13_UpDownBack : BOOL;
    SOL_S13_UpDown : BOOL;
    LS_S15_UpDownBack : BOOL;
    SOL_S15_UpDown : BOOL;
END_VAR
(*************************************************************************
程序名稱:轉盤程式
作者:蔡相偉
版本,日期,版本資訊:
1.0.0	2017/8/8		初始版本
流程
PowerOn=0
Idle=1
轉盤定位回=2
轉盤起動=3
轉盤運轉中=4
轉盤停止=5
轉盤定位出=6
*************************************************************************)
(*PowerOn=0*)
IF NOT(SystemReadyStatus) OR ErrorStatus[0] THEN
	AutoFlow:=0;
END_IF;
(*Idle=1*)
IF AutoFlow=0 AND SystemReadyStatus AND NOT(ErrorStatus[0]) THEN
	AutoFlow:=1;
END_IF;
IF Autoflow=6 AND TON_1.Q THEN
	Autoflow:=1;
END_IF;
(*轉盤定位回=2*)
R_TRIG_1(CLK:= HMIPB_RY_Index AND NOT(AutoStatus));
IF Autoflow=1 AND IndexCanRunStatus AND (R_TRIG_1.Q OR
	(MachineRunStatus AND
	IndexData[1].FinishFlag[1] AND
	IndexData[2].FinishFlag[2] AND
	IndexData[4].FinishFlag[4] AND
	IndexData[5].FinishFlag[5] AND
	IndexData[6].FinishFlag[6] AND
	IndexData[7].FinishFlag[7] AND
	IndexData[8].FinishFlag[8] AND
	IndexData[9].FinishFlag[9] AND
	IndexData[10].FinishFlag[10] AND
	IndexData[11].FinishFlag[11] AND
	IndexData[13].FinishFlag[13] AND
	IndexData[15].FinishFlag[15] AND
	IndexData[16].FinishFlag[16])) THEN
	Autoflow:=2;
END_IF;

(*轉盤起動=3*)
IF Autoflow=2 THEN
	Autoflow:=3;
END_IF;

(*轉盤運轉中=4*)
IF Autoflow=3 AND NOT(SNR_Index) THEN
	Autoflow:=4;
END_IF;

(*轉盤停止=5*)
IF Autoflow=4 AND SNR_Index THEN
	Autoflow:=5;
END_IF;

(*轉盤定位出=6*)
IF Autoflow=5 THEN
	Autoflow:=6;
END_IF;
tDelayTime:=NanoSecToTime(HMISV_Index_DelayTime*100000);
TON_1(IN:= Autoflow=6 ,PT:= tDelayTime);

(******************************************************************)
(*輸出*)
IndexCanRunStatus:=
YAMAHA_ORG AND
(LS_S2_UpDownBack AND NOT(SOL_S2_UpDown)) AND
((LS_S4_UpDownBack AND NOT(SOL_S4_UpDown)) OR NOT(LS_S4_MoveBack)) AND
((LS_S6_UpDownBack AND NOT(SOL_S6_UpDown)) OR NOT(LS_S6_MoveBack)) AND
((LS_S8_UpDownBack AND NOT(SOL_S8_UpDown)) OR NOT(LS_S8_MoveOut)) AND
((LS_S10_UpDownBack AND NOT(SOL_S10_UpDown)) OR NOT(LS_S10_MoveOut)) AND
(LS_S11_UpDownBack AND NOT(SOL_S11_UpDown)) AND
(LS_S13_UpDownBack AND NOT(SOL_S13_UpDown)) AND
(LS_S15_UpDownBack AND NOT(SOL_S15_UpDown));

(*轉盤運轉*)
IF (AutoFlow=3 OR Autoflow=4) AND IndexCanRunStatus THEN
	RY_Index:=TRUE;
	ELSE
	RY_Index:=FALSE;
END_IF;
END_PROGRAM

PROGRAM prStation1_PanelLoad
VAR
    Autoflow : INT;
    Initflow : INT;
    interlockback : ARRAY[0..2] OF BOOL;
    interlockout : ARRAY[0..2] OF BOOL;
    solStatus : ARRAY[0..2] OF BOOL;
    R_TRIG_1 : ARRAY[0..2] OF R_TRIG;
    F_TRIG_1 : F_TRIG;
    ErrorLS : BOOL;
    StartFlag : BOOL;
    TON_1 : TON;
    TON_2 : TON;
    TON_3 : TON;
END_VAR
VAR_EXTERNAL
    HMIPB_SOL_S1_Load_PanelUpDown1Back : BOOL;
    SOL_S1_Load_PanelUpDown1Back : BOOL;
    SOL_S1_Load_PanelUpDown1Out : BOOL;
    LS_S1_Load_PanelUpDown1Back : BOOL;
    HMIPB_SOL_S1_Load_PanelUpDown1Out : BOOL;
    AutoStatus : BOOL;
    LS_S1_Load_PanelUpDown1Out : BOOL;
    HMIPB_SOL_S1_Load_PanelUpDown2Back : BOOL;
    SOL_S1_Load_PanelUpDown2Back : BOOL;
    SOL_S1_Load_PanelUpDown2Out : BOOL;
    LS_S1_Load_PanelUpDown2Back : BOOL;
    HMIPB_SOL_S1_Load_PanelUpDown2Out : BOOL;
    LS_S1_Load_PanelUpDown2Out : BOOL;
    HMIPB_SOL_S1_Load_PanelClip : BOOL;
    SOL_S1_Load_PanelClip : BOOL;
    SystemReadyStatus : BOOL;
    ErrorStatus : ARRAY[0..19] OF BOOL;
    Error_PB_EStop : BOOL;
    SNR_S1_Load_PanelFeed : BOOL;
    LS_S1_Load_PanelClip1Out : BOOL;
    LS_S1_Load_PanelClip2Out : BOOL;
    LS_S1_Load_PanelClip2Back : BOOL;
    LS_S1_Load_PanelClip1Back : BOOL;
    RY_S1_Load_VariableSpeedMotor : BOOL;
    Error_LS_S1_Load_PanelUpDown1Back : BOOL;
    Error_LS_S1_Load_PanelUpDown1Out : BOOL;
    Error_LS_S1_Load_PanelUpDown2Back : BOOL;
    Error_LS_S1_Load_PanelUpDown2Out : BOOL;
    Error_LS_S1_Load_PanelClip1Back : BOOL;
    Error_LS_S1_Load_PanelClip1Out : BOOL;
    Error_LS_S1_Load_PanelClip2Back : BOOL;
    Error_LS_S1_Load_PanelClip2Out : BOOL;
    ErrorStatus_S1_Load : BOOL;
END_VAR
(*
程序名稱: Panel LOAD程序
作者:蔡相偉
版本,日期,版本資訊:
1.0.0		2017/11/16		初始版本

PowerOn=0
Idle=1
Panel出盤程序開始=10
第1段,第2段出=2
夾持出=3
第2段回=4
夾持回=5
第1段回=6
*)
//***************************************************************************************************************
//Define
ErrorLS:=ErrorStatus_S1_Load;
StartFlag:=TON_1.Q;
TON_1(In:=NOT(SNR_S1_Load_PanelFeed) AND NOT(RY_S1_Load_VariableSpeedMotor), PT:=t#5s);
//PowerOn=0
IF NOT(SystemReadyStatus AND NOT(ErrorLS) AND  NOT(Error_PB_Estop) AND AutoStatus) THEN
	Autoflow:=0;
END_IF;

//Idle=1
IF AutoFlow=0 AND SystemReadyStatus AND NOT(ErrorLS) AND  NOT(Error_PB_Estop) AND AutoStatus THEN
	AutoFlow:=1;
END_IF;

IF Autoflow=6 AND LS_S1_Load_PanelUpDown1Back THEN
	Autoflow:=1;
END_IF;

//第1段,第2段出=2
IF Autoflow=1 AND StartFlag THEN
	Autoflow:=2;
END_IF;

//承盤夾持出=3
IF Autoflow=2 AND LS_S1_Load_PanelUpDown1Out AND LS_S1_Load_PanelUpDown2Out THEN
	Autoflow:=3;
END_IF;
TON_2(In:= Autoflow=3 AND LS_S1_Load_PanelClip1Out AND LS_S1_Load_PanelClip2Out , PT:=t#300ms);

//第2段回=4
IF Autoflow=3 AND TON_2.Q THEN
	Autoflow:=4;
END_IF;
TON_3(In:=Autoflow=4 AND LS_S1_Load_PanelUpDown2Back, PT:=t#300ms);

//承盤夾持回=5
IF Autoflow=4 AND TON_3.Q THEN
	Autoflow:=5;
END_IF;

//第1段回=6
IF Autoflow=5 AND  LS_S1_Load_PanelClip1Back AND LS_S1_Load_PanelClip2Back THEN
	Autoflow:=6;
END_IF;

//***************************************************************************************************************
//下夾板出盤下降第1段回電磁閥
interlockback[0]:=NOT(RY_S1_Load_VariableSpeedMotor);
IF ((HMIPB_SOL_S1_Load_PanelUpDown1Back AND NOT(AutoStatus)) OR Autoflow=6 OR Initflow=6) AND interlockback[0] THEN
	SOL_S1_Load_PanelUpDown1Back:=TRUE;
	SOL_S1_Load_PanelUpDown1Out:=FALSE;
END_IF;
IF LS_S1_Load_PanelUpDown1Back THEN
	SOL_S1_Load_PanelUpDown1Back:=FALSE;
END_IF;

//下夾板出盤下降第1段出電磁閥
interlockout[0]:=TRUE;
IF ((HMIPB_SOL_S1_Load_PanelUpDown1Out AND NOT(AutoStatus)) OR Autoflow=2) AND interlockout[0] THEN
	SOL_S1_Load_PanelUpDown1Back:=FALSE;
	SOL_S1_Load_PanelUpDown1Out:=TRUE;
END_IF;
IF LS_S1_Load_PanelUpDown1Out THEN
	SOL_S1_Load_PanelUpDown1Out:=FALSE;
END_IF;
//***************************************************************************************************************
//下夾板出盤下降第2段回電磁閥
interlockback[1]:=TRUE;
IF ((HMIPB_SOL_S1_Load_PanelUpDown2Back AND NOT(AutoStatus)) OR Autoflow=4 OR Initflow=4) AND interlockback[1] THEN
	SOL_S1_Load_PanelUpDown2Back:=TRUE;
	SOL_S1_Load_PanelUpDown2Out:=FALSE;
END_IF;
IF LS_S1_Load_PanelUpDown2Back THEN
	SOL_S1_Load_PanelUpDown2Back:=FALSE;
END_IF;

//下夾板出盤下降第2段出電磁閥
interlockout[1]:=TRUE;
IF ((HMIPB_SOL_S1_Load_PanelUpDown2Out AND NOT(AutoStatus)) OR Autoflow=2) AND interlockout[1] THEN
	SOL_S1_Load_PanelUpDown2Back:=FALSE;
	SOL_S1_Load_PanelUpDown2Out:=TRUE;
END_IF;
IF LS_S1_Load_PanelUpDown2Out THEN
	SOL_S1_Load_PanelUpDown2Out:=FALSE;
END_IF;
//***************************************************************************************************************
(*下夾板出盤承載電磁閥*)
R_TRIG_1[2](CLK:=HMIPB_SOL_S1_Load_PanelClip AND NOT(AutoStatus));
interlockback[2]:=TRUE;
interlockout[2]:=LS_S1_Load_PanelUpDown1Out;
(*SET*)
IF ((R_TRIG_1[2].Q AND NOT(solStatus[2])) OR Autoflow=3) AND interlockout[2] THEN
	SOL_S1_Load_PanelClip:=TRUE;
END_IF;
(*RESET*)
IF ((R_TRIG_1[2].Q AND (solStatus[2])) OR Autoflow=5 OR Initflow=5) AND interlockback[2] THEN
	SOL_S1_Load_PanelClip:=FALSE;
END_IF;
(*STATUS*)
solStatus[2]:=SOL_S1_Load_PanelClip;

//***************************************************************************************************************
(*
程序名稱: Panel LOAD RESET程序
作者:蔡相偉
版本,日期,版本資訊:
1.0.0		2017/11/16		初始版本

PowerOn=0
Idle=1
第2段回=4
夾持回=5
第1段回=6

//***************************************************************************************************************
//PowerOn=0
IF NOT(SystemReadyStatus) THEN
	Initflow:=0;
END_IF;

//Idle=1
IF Initflow=0 AND SystemReadyStatus THEN
	Initflow:=1;
END_IF;

IF Initflow=6 AND LS_S1_Load_PanelUpDown1Back THEN
	Initflow:=1;
END_IF;

F_TRIG_1(Clk:=ErrorLS);
//第2段回=4
IF Initflow=1 AND F_TRIG_1.Q THEN
	Initflow:=4;
END_IF;

//承盤夾持回=5
IF Initflow=4 AND LS_S1_Load_PanelUpDown2Back THEN
	Initflow:=5;
END_IF;

//第1段回=6
IF Initflow=5 AND  LS_S1_Load_PanelClip1Back AND LS_S1_Load_PanelClip2Back THEN
	Initflow:=6;
END_IF;
*)
END_PROGRAM

PROGRAM prStation1_FeedPanelLoad
VAR
    Autoflow : INT;
    interlockback : ARRAY[0..3] OF BOOL;
    interlockout : ARRAY[0..3] OF BOOL;
    solStatus : ARRAY[0..3] OF BOOL;
    R_TRIG_1 : ARRAY[0..3] OF R_TRIG;
    ErrorLS : BOOL;
    StartFlag : BOOL;
    TON_1 : TON;
    TON_2 : TON;
    TON_3 : TON;
    TON_4 : TON;
    TON_5 : TON;
    TON_6 : TON;
    F_TRIG_1 : F_TRIG;
    centermotorStartflag : BOOL;
END_VAR
VAR_EXTERNAL
    HMIPB_SOL_S1_Load_PanelUpDown1Back : BOOL;
    SOL_S1_Load_PanelUpDown1Back : BOOL;
    SOL_S1_Load_PanelUpDown1Out : BOOL;
    LS_S1_Load_PanelUpDown1Back : BOOL;
    HMIPB_SOL_S1_Load_PanelUpDown1Out : BOOL;
    AutoStatus : BOOL;
    LS_S1_Load_PanelUpDown1Out : BOOL;
    HMIPB_SOL_S1_Load_PanelUpDown2Back : BOOL;
    SOL_S1_Load_PanelUpDown2Back : BOOL;
    SOL_S1_Load_PanelUpDown2Out : BOOL;
    LS_S1_Load_PanelUpDown2Back : BOOL;
    HMIPB_SOL_S1_Load_PanelUpDown2Out : BOOL;
    LS_S1_Load_PanelUpDown2Out : BOOL;
    HMIPB_SOL_S1_Load_PanelClip : BOOL;
    SOL_S1_Load_PanelClip : BOOL;
    HMIPB_SOL_S1_Load_FixClip : BOOL;
    SOL_S1_Load_FixClip : BOOL;
    HMIPB_SOL_S1_Load_ConveyorClip : BOOL;
    SOL_S1_Load_ConveyorClip : BOOL;
    HMIPB_SOL_S1_Load_UpDown : BOOL;
    SOL_S1_Load_UpDown : BOOL;
    HMIPB_RY_S1_Load_VariableSpeedMotor : BOOL;
    RY_S1_Load_VariableSpeedMotor : BOOL;
    RY_S1_Load_FixSpeedMotor : BOOL;
    HMIPB_RY_S1_Load_FixSpeedMotor : BOOL;
    SNR_S1_Load_PanelFeed : BOOL;
    SNR_S1_Load_PanelClip : BOOL;
    SystemReadyStatus : BOOL;
    ErrorStatus : ARRAY[0..19] OF BOOL;
    ErrorStatus_TH : ARRAY[0..19] OF BOOL;
    RY_S1_Center_VariableSpeedMotor : BOOL;
    HMIPB_RY_S1_Center_VariableSpeedMotor : BOOL;
    Error_PB_EStop : BOOL;
    ErrorStatus_S1_FeedPanelLoad : BOOL;
    HMIPB_SOL_S1_Load_AlignmentClip : BOOL;
    SOL_S1_Load_AlignmentClip : BOOL;
    YAMAHA_Load_ChangePanelStart : BOOL;
    HMIPB_YAMAHA_Load_ChangePanelStart : BOOL;
    SNR_AirSource : BOOL;
    SNR_S1_Load_Feed : BOOL;
    SNR_S1_UnLoad_Feed : BOOL;
    LS_S1_Load_FixClipOut : BOOL;
    LS_S1_Load_AlignmentClipOut : BOOL;
    HMIPB_YAMAHA_Unload_ChangePanelStart : BOOL;
    LS_S1_Load_UpDownOut : BOOL;
    LS_S1_Load_ConveyorClip1Out : BOOL;
    LS_S1_Load_ConveyorClip2Out : BOOL;
    LS_S10_ClipFBack : BOOL;
    LS_S1_Load_UpDownBack : BOOL;
    LS_S1_Load_ConveyorClip1Back : BOOL;
    LS_S1_Load_ConveyorClip2Back : BOOL;
    LS_S1_Load_FixClipBack : BOOL;
    LS_S1_Load_AlignmentClipBack : BOOL;
    YAMAHA_Load_Ready : BOOL;
    YAMAHA_Load_Finish : BOOL;
    YAMAHA_Load_Start : BOOL;
    YAMAHA_Unload_ChangePanelStart : BOOL;
END_VAR
(*
程序名稱: 出盤程序
作者:蔡相偉
版本,日期,版本資訊:
1.0.0		2017/11/16		初始版本

PowerOn=0--->
Idle=1--->
換盤程序開始=2|--->工件取放處有盤=10--->固定,活動夾持出=11--->上下出=12--->軌道夾持出=13--->上下回=14--->軌道夾持回=15--->20
						  |--->工件取放處無盤=20--->軌道夾持回=21--->固定,活動夾持出=22--->馬達ON=23--->馬達運行中=24--->盤到位,馬達停止=25--->固定邊夾持回=26--->活動邊夾持回=27--->換盤完成=28--->1
*)
(*
Error Code
1:緊急停止
2:磁簧異常
*)
//***************************************************************************************************************
//Define
ErrorLS:=
ErrorStatus_S1_FeedPanelLoad;
//***************************************************************************************************************
//PowerOn=0
IF NOT(SystemReadyStatus AND NOT(ErrorLS) AND  NOT(Error_PB_Estop) AND AutoStatus) THEN
	Autoflow:=0;
END_IF;

//Idle=1
IF Autoflow=0 AND SystemReadyStatus AND NOT(ErrorLS) AND  NOT(Error_PB_Estop) AND AutoStatus THEN
	Autoflow:=1;
END_IF;

IF Autoflow=28 AND NOT(YAMAHA_Load_ChangePanelStart) THEN
	Autoflow:=1;
END_IF;

TON_1(In:=Autoflow=1 AND NOT(SNR_S1_Load_PanelClip), PT:=t#1s);

IF Autoflow=1 AND TON_5.Q THEN		(*READY訊號*)
	YAMAHA_Load_Ready:=TRUE;
ELSE
	YAMAHA_Load_Ready:=FALSE;
END_IF;

//換盤程序開始=2
IF Autoflow=1 AND (YAMAHA_Load_ChangePanelStart OR HMIPB_YAMAHA_Load_ChangePanelStart OR TON_1.Q) THEN
	Autoflow:=2;
END_IF;

//工件取放處有盤=10
IF Autoflow=2 AND SNR_S1_Load_PanelClip THEN
	Autoflow:=10;
END_IF;

//固定,活動夾持出=11
IF Autoflow=10 THEN
	Autoflow:=11;
END_IF;
IF Autoflow=11 AND SNR_S1_Load_Feed THEN
	HMIPB_YAMAHA_Unload_ChangePanelStart:=TRUE;
END_IF;

//上下出=12
IF Autoflow=11 AND LS_S1_Load_FixClipOut AND LS_S1_Load_AlignmentClipOut AND TON_4.Q THEN
	Autoflow:=12;
END_IF;

//軌道夾持出=13
IF Autoflow=12 AND LS_S1_Load_UpDownOut THEN
	Autoflow:=13;
END_IF;

//上下回=14
IF Autoflow=13 AND LS_S1_Load_ConveyorClip1Out AND LS_S1_Load_ConveyorClip2Out THEN
	Autoflow:=14;
END_IF;

//軌道夾持回=15
IF Autoflow=14 AND LS_S1_Load_UpDownBack THEN
	Autoflow:=15;
END_IF;
//***************************************************************************************************************
//工件取放處無盤=20
IF Autoflow=2 AND NOT(SNR_S1_Load_PanelClip) THEN
	Autoflow:=20;
END_IF;

IF Autoflow=15 AND LS_S1_Load_ConveyorClip1Back AND LS_S1_Load_ConveyorClip2Back THEN
	Autoflow:=20;
END_IF;

//軌道夾持回=21
IF Autoflow=20 THEN
	Autoflow:=21;
END_IF;

//固定,活動夾持出=22
IF Autoflow=21 AND LS_S1_Load_ConveyorClip1Back AND LS_S1_Load_ConveyorClip2Back THEN
	Autoflow:=22;
END_IF;

//馬達ON=23
IF Autoflow=22 AND LS_S1_Load_FixClipOut AND LS_S1_Load_AlignmentClipOut AND SNR_S1_Load_PanelFeed THEN
	Autoflow:=23;
END_IF;
IF Autoflow=23 THEN
	HMIPB_RY_S1_Load_FixSpeedMotor:=TRUE;
	HMIPB_RY_S1_Load_VariableSpeedMotor:=TRUE;
END_IF;

//馬達運行中=24
IF Autoflow=23 AND RY_S1_Load_FixSpeedMotor AND RY_S1_Load_VariableSpeedMotor THEN
	Autoflow:=24;
END_IF;


//盤到位,馬達停止=25
IF Autoflow=24 AND TON_5.Q THEN
	Autoflow:=25;
END_IF;


//固定邊夾持回=26
IF Autoflow=25 AND NOT(RY_S1_Load_FixSpeedMotor) AND NOT(RY_S1_Load_VariableSpeedMotor) THEN
	Autoflow:=26;
END_IF;

//活動邊夾持回=27
IF Autoflow=26 AND LS_S1_Load_FixClipBack THEN
	Autoflow:=27;
END_IF;
//換盤完成=28
IF Autoflow=27 AND LS_S1_Load_AlignmentClipBack THEN
	Autoflow:=28;
END_IF;

//***************************************************************************************************************
//下夾板出盤固定邊定位電磁閥
R_TRIG_1[0](CLK:=HMIPB_SOL_S1_Load_FixClip AND NOT(AutoStatus));
interlockback[0]:=TRUE;
interlockout[0]:=TRUE;
//SET
IF ((R_TRIG_1[0].Q AND NOT(solStatus[0])) OR Autoflow=11 OR Autoflow=22) AND interlockout[0] THEN
	SOL_S1_Load_FixClip:=TRUE;
END_IF;
//RESET
IF ((R_TRIG_1[0].Q AND (solStatus[0])) OR Autoflow=26) AND interlockback[0] THEN
	SOL_S1_Load_FixClip:=FALSE;
END_IF;
//STATUS
solStatus[0]:=SOL_S1_Load_FixClip;
//***************************************************************************************************************
//下夾板出盤活動邊定位電磁閥
R_TRIG_1[1](CLK:=HMIPB_SOL_S1_Load_AlignmentClip AND NOT(AutoStatus));
interlockback[1]:=TRUE;
interlockout[1]:=TRUE;
//SET
IF ((R_TRIG_1[1].Q AND NOT(solStatus[1])) OR Autoflow=11 OR Autoflow=22) AND interlockout[1] THEN
	SOL_S1_Load_AlignmentClip:=TRUE;
END_IF;
//RESET
IF ((R_TRIG_1[1].Q AND (solStatus[1])) OR Autoflow=27) AND interlockback[1] THEN
	SOL_S1_Load_AlignmentClip:=FALSE;
END_IF;
//STATUS
solStatus[1]:=SOL_S1_Load_AlignmentClip;
//***************************************************************************************************************
//下夾板出盤軌道開合電磁閥
R_TRIG_1[2](CLK:=HMIPB_SOL_S1_Load_ConveyorClip AND NOT(AutoStatus));
interlockback[2]:=TRUE;
interlockout[2]:=LS_S1_Load_UpDownOut AND SOL_S1_Load_UpDown;
//SET
IF ((R_TRIG_1[2].Q AND NOT(solStatus[2])) OR Autoflow=13) AND interlockout[2] THEN
	SOL_S1_Load_ConveyorClip:=TRUE;
END_IF;
//RESET
IF ((R_TRIG_1[2].Q AND (solStatus[2])) OR Autoflow=15 OR Autoflow=21) AND interlockback[2] THEN
	SOL_S1_Load_ConveyorClip:=FALSE;
END_IF;
//STATUS
solStatus[2]:=SOL_S1_Load_ConveyorClip;
//***************************************************************************************************************
//下夾板出盤升降電磁閥
R_TRIG_1[3](CLK:=HMIPB_SOL_S1_Load_UpDown AND NOT(AutoStatus));
interlockback[3]:=TRUE;
interlockout[3]:=LS_S1_Load_AlignmentClipOut AND SOL_S1_Load_AlignmentClip AND LS_S1_Load_FixClipOut AND SOL_S1_Load_FixClip;
//RESET
IF ((R_TRIG_1[3].Q AND NOT(solStatus[3])) OR Autoflow=12) AND interlockout[3] THEN
	SOL_S1_Load_UpDown:=TRUE;
END_IF;
//RESET
IF ((R_TRIG_1[3].Q AND (solStatus[3])) OR Autoflow=14) AND interlockback[3] THEN
	SOL_S1_Load_UpDown:=FALSE;
END_IF;
//STATUS
solStatus[3]:=SOL_S1_Load_UpDown;
//***************************************************************************************************************
//下夾板出盤調速馬達繼電器
//RESET
TON_6(In:=NOT(SNR_S1_Load_PanelFeed), PT:=t#1s);
IF TON_6.Q THEN
	HMIPB_RY_S1_Load_VariableSpeedMotor:=FALSE;
END_IF;
//OUT
RY_S1_Load_VariableSpeedMotor:=HMIPB_RY_S1_Load_VariableSpeedMotor;
//***************************************************************************************************************
//下夾板出盤定速馬達繼電器
//RESET
TON_5(In:=SNR_S1_Load_PanelClip, PT:=t#1s);
IF TON_5.Q THEN
	HMIPB_RY_S1_Load_FixSpeedMotor:=FALSE;
END_IF;
//OUT
RY_S1_Load_FixSpeedMotor:=HMIPB_RY_S1_Load_FixSpeedMotor;
//***************************************************************************************************************
//下夾板下移載調速馬達繼電器
TON_2(In:=SNR_S1_Load_Feed, PT:=t#1s);
IF TON_2.Q OR HMIPB_RY_S1_Center_VariableSpeedMotor OR ((HMIPB_YAMAHA_Unload_ChangePanelStart OR YAMAHA_Unload_ChangePanelStart) AND NOT(SNR_S1_UnLoad_Feed)) THEN
	centermotorStartflag:=TRUE;
END_IF;
TON_3(In:=not(SNR_S1_Load_Feed), PT:=t#500ms);
IF TON_3.Q AND NOT(HMIPB_RY_S1_Center_VariableSpeedMotor) AND NOT((HMIPB_YAMAHA_Unload_ChangePanelStart OR YAMAHA_Unload_ChangePanelStart) AND NOT(SNR_S1_UnLoad_Feed)) THEN
	centermotorStartflag:=FALSE;
END_IF;

//OUT
RY_S1_Center_VariableSpeedMotor:=centermotorStartflag;
END_PROGRAM

PROGRAM prError
VAR
    TON_1 : TON;
    ErrorDouble : ARRAY[0..30] of fbErrorDouble;
    ErrorSingle : ARRAY[0..30] of fbErrorSingle;
END_VAR
VAR_EXTERNAL
    IndexData : ARRAY[0..19] OF stIndexData;
    ErrorStatus_TH : ARRAY[0..19] OF BOOL;
    SystemReadyStatus : BOOL;
    PB_Estop : BOOL;
    Error_PB_Estop : BOOL;
    RY_Index : BOOL;
    Error_SNR_index : BOOL;
    SNR_AirSource : BOOL;
    Error_SNR_AirSource : BOOL;
    Invertor_Ready : BOOL;
    Error_Invertor_Ready : BOOL;
    AutoStatus : BOOL;
    PB_Reset : BOOL;
    LS_S1_Load_PanelUpDown1Back : BOOL;
    LS_S1_Load_PanelUpDown1Out : BOOL;
    SOL_S1_Load_PanelUpDown1Back : BOOL;
    SOL_S1_Load_PanelUpDown1Out : BOOL;
    Error_LS_S1_Load_PanelUpDown1Back : BOOL;
    Error_LS_S1_Load_PanelUpDown1Out : BOOL;
    LS_S1_Load_PanelUpDown2Back : BOOL;
    LS_S1_Load_PanelUpDown2Out : BOOL;
    SOL_S1_Load_PanelUpDown2Back : BOOL;
    SOL_S1_Load_PanelUpDown2Out : BOOL;
    Error_LS_S1_Load_PanelUpDown2Back : BOOL;
    Error_LS_S1_Load_PanelUpDown2Out : BOOL;
    ErrorStatus_MachineStop : BOOL;
    ErrorStatus : ARRAY[0..19] OF BOOL;
    ErrorStatus_MachineNonStop : BOOL;
    ErrorStatus_MachineStop_Record : BOOL;
    ErrorStatus_S1_Load : BOOL;
    LS_S1_Load_PanelClip1Back : BOOL;
    LS_S1_Load_PanelClip1Out : BOOL;
    SOL_S1_Load_PanelClip : BOOL;
    Error_LS_S1_Load_PanelClip1Back : BOOL;
    Error_LS_S1_Load_PanelClip1Out : BOOL;
    LS_S1_Load_PanelClip2Back : BOOL;
    LS_S1_Load_PanelClip2Out : BOOL;
    Error_LS_S1_Load_PanelClip2Back : BOOL;
    Error_LS_S1_Load_PanelClip2Out : BOOL;
    ErrorStatus_S1_UnLoad : BOOL;
    LS_S1_Load_FixClipBack : BOOL;
    LS_S1_Load_FixClipOut : BOOL;
    SOL_S1_Load_FixClip : BOOL;
    Error_LS_S1_Load_FixClipBack : BOOL;
    Error_LS_S1_Load_FixClipOut : BOOL;
    ErrorStatus_S1_FeedPanelLoad : BOOL;
    LS_S1_Load_ConveyorClip1Back : BOOL;
    LS_S1_Load_ConveyorClip1Out : BOOL;
    SOL_S1_Load_ConveyorClip : BOOL;
    Error_LS_S1_Load_ConveyorClip1Back : BOOL;
    Error_LS_S1_Load_ConveyorClip1Out : BOOL;
    LS_S1_Load_AlignmentClipBack : BOOL;
    LS_S1_Load_AlignmentClipOut : BOOL;
    SOL_S1_Load_AlignmentClip : BOOL;
    Error_LS_S1_Load_AlignmentClipBack : BOOL;
    Error_LS_S1_Load_AlignmentClipOut : BOOL;
    LS_S1_Load_UpDownBack : BOOL;
    LS_S1_Load_UpDownOut : BOOL;
    SOL_S1_Load_UpDown : BOOL;
    Error_LS_S1_Load_UpDownBack : BOOL;
    Error_LS_S1_Load_UpDownOut : BOOL;
    ErrorStatus_S1_FeedPanelUnLoad : BOOL;
    LS_S1_UnLoad_PanelUpDown1Back : BOOL;
    LS_S1_UnLoad_PanelUpDown1Out : BOOL;
    SOL_S1_UnLoad_PanelUpDown1Back : BOOL;
    SOL_S1_UnLoad_PanelUpDown1Out : BOOL;
    Error_LS_S1_UnLoad_PanelUpDown1Back : BOOL;
    Error_LS_S1_UnLoad_PanelUpDown1Out : BOOL;
    LS_S1_UnLoad_PanelUpDown2Back : BOOL;
    LS_S1_UnLoad_PanelUpDown2Out : BOOL;
    SOL_S1_UnLoad_PanelUpDown2Back : BOOL;
    SOL_S1_UnLoad_PanelUpDown2Out : BOOL;
    Error_LS_S1_UnLoad_PanelUpDown2Back : BOOL;
    Error_LS_S1_UnLoad_PanelUpDown2Out : BOOL;
    LS_S1_UnLoad_PanelClip1Back : BOOL;
    LS_S1_UnLoad_PanelClip1Out : BOOL;
    SOL_S1_UnLoad_PanelClip : BOOL;
    Error_LS_S1_UnLoad_PanelClip1Back : BOOL;
    Error_LS_S1_UnLoad_PanelClip1Out : BOOL;
    LS_S1_UnLoad_PanelClip2Back : BOOL;
    LS_S1_UnLoad_PanelClip2Out : BOOL;
    SOL_S1_UnLoad_FixClip : BOOL;
    Error_LS_S1_UnLoad_PanelClip2Back : BOOL;
    Error_LS_S1_UnLoad_PanelClip2Out : BOOL;
    LS_S1_UnLoad_FixClipBack : BOOL;
    LS_S1_UnLoad_FixClipOut : BOOL;
    Error_LS_S1_UnLoad_FixClipBack : BOOL;
    Error_LS_S1_UnLoad_FixClipOut : BOOL;
    LS_S1_UnLoad_AlignmentClipBack : BOOL;
    LS_S1_UnLoad_AlignmentClipOut : BOOL;
    SOL_S1_UnLoad_AlignmentClip : BOOL;
    Error_LS_S1_UnLoad_AlignmentClipBack : BOOL;
    Error_LS_S1_UnLoad_AlignmentClipOut : BOOL;
    LS_S1_UnLoad_ConveyorClip1Back : BOOL;
    LS_S1_UnLoad_ConveyorClip1Out : BOOL;
    SOL_S1_UnLoad_ConveyorClip : BOOL;
    Error_LS_S1_UnLoad_ConveyorClip1Back : BOOL;
    Error_LS_S1_UnLoad_ConveyorClip1Out : BOOL;
    LS_S1_UnLoad_UpDownBack : BOOL;
    LS_S1_UnLoad_UpDownOut : BOOL;
    SOL_S1_UnLoad_UpDown : BOOL;
    Error_LS_S1_UnLoad_UpDownBack : BOOL;
    Error_LS_S1_UnLoad_UpDownOut : BOOL;
    Error_SNR_S10_Full : BOOL;
    Error_SNR_S1_Load_Full : BOOL;
    Error_SNR_S1_UnLoad_Full : BOOL;
    Error_SNR_S4_Load_Full : BOOL;
    Error_SNR_S4_UnLoad_Full : BOOL;
    Error_SNR_S6_Full : BOOL;
    Error_SNR_S8_Full : BOOL;
    YAMAHA_S_State_Alarm : BOOL;
    YAMAHA_S_State_Warring : BOOL;
    YAMAHA_Error_SOL_Clip : BOOL;
END_VAR
(*緊急停止*)
(*
IF SystemReadyStatus AND NOT(PB_Estop) THEN
	Error_PB_Estop:=TRUE;
END_IF;
*)
//**********************************************************************************************************************
(*轉盤微動開關*)
TON_1(IN:= RY_Index ,PT:= t#6s);
IF TON_1.Q THEN
	Error_SNR_index:=TRUE;
END_IF;
//**********************************************************************************************************************
(*總氣源*)
IF SystemReadyStatus AND NOT(SNR_AirSource) THEN
	Error_SNR_AirSource:=TRUE;
END_IF;
//**********************************************************************************************************************
(*變頻器*)
IF SystemReadyStatus AND Invertor_Ready THEN
	Error_Invertor_Ready:=TRUE;
END_IF;
//**********************************************************************************************************************
//**********************************************************************************************************************
//Station0
//**********************************************************************************************************************
(*異常*)
ErrorStatus[0]:=
Error_PB_Estop OR
Error_SNR_index OR
Error_SNR_AirSource OR
Error_Invertor_Ready;
//**********************************************************************************************************************
(*Station1*)
//**********************************************************************************************************************
//LOAD
ErrorDouble[0](
	bAutoStatus:=AutoStatus,
	bResetPB:=PB_Reset,
	bBackLS:=LS_S1_Load_PanelUpDown1Back, bOutLS:=LS_S1_Load_PanelUpDown1Out,
	bBackSOL:=SOL_S1_Load_PanelUpDown1Back, bOutSOL:=SOL_S1_Load_PanelUpDown1Out,
	bErrorStatus_Back=>Error_LS_S1_Load_PanelUpDown1Back, bErrorStatus_Out=>Error_LS_S1_Load_PanelUpDown1Out);

ErrorDouble[1](
	bAutoStatus:=AutoStatus,
	bResetPB:=PB_Reset,
	bBackLS:=LS_S1_Load_PanelUpDown2Back, bOutLS:=LS_S1_Load_PanelUpDown2Out,
	bBackSOL:=SOL_S1_Load_PanelUpDown2Back,
	bOutSOL:=SOL_S1_Load_PanelUpDown2Out,
	bErrorStatus_Back=>Error_LS_S1_Load_PanelUpDown2Back,
	bErrorStatus_Out=>Error_LS_S1_Load_PanelUpDown2Out);

ErrorSingle[0](
	bAutoStatus:=AutoStatus,
	bResetPB:=PB_Reset,
	bBackLS:=LS_S1_Load_PanelClip1Back,
	bOutLS:=LS_S1_Load_PanelClip1Out,
	bSOL:=SOL_S1_Load_PanelClip,
	bErrorStatus_Back=>Error_LS_S1_Load_PanelClip1Back,
	bErrorStatus_Out=>Error_LS_S1_Load_PanelClip1Out);

ErrorSingle[1](
	bAutoStatus:=AutoStatus,
	bResetPB:=PB_Reset,
	bBackLS:=LS_S1_Load_PanelClip2Back,
	bOutLS:=LS_S1_Load_PanelClip2Out,
	bSOL:=SOL_S1_Load_PanelClip,
	bErrorStatus_Back=>Error_LS_S1_Load_PanelClip2Back,
	bErrorStatus_Out=>Error_LS_S1_Load_PanelClip2Out);

//Load 後段
ErrorSingle[2](
	bAutoStatus:=AutoStatus,
	bResetPB:=PB_Reset,
	bBackLS:=LS_S1_Load_FixClipBack,
	bOutLS:=LS_S1_Load_FixClipOut,
	bSOL:=SOL_S1_Load_FixClip,
	bErrorStatus_Back=>Error_LS_S1_Load_FixClipBack,
	bErrorStatus_Out=>Error_LS_S1_Load_FixClipOut);

ErrorSingle[3](
	bAutoStatus:=AutoStatus,
	bResetPB:=PB_Reset,
	bBackLS:=LS_S1_Load_AlignmentClipBack,
	bOutLS:=LS_S1_Load_AlignmentClipOut,
	bSOL:=SOL_S1_Load_AlignmentClip,
	bErrorStatus_Back=>Error_LS_S1_Load_AlignmentClipBack,
	bErrorStatus_Out=>Error_LS_S1_Load_AlignmentClipOut);

ErrorSingle[4](
	bAutoStatus:=AutoStatus,
	bResetPB:=PB_Reset,
	bBackLS:=LS_S1_Load_ConveyorClip1Back,
	bOutLS:=LS_S1_Load_ConveyorClip1Out,
	bSOL:=SOL_S1_Load_ConveyorClip,
	bErrorStatus_Back=>Error_LS_S1_Load_ConveyorClip1Back,
	bErrorStatus_Out=>Error_LS_S1_Load_ConveyorClip1Out);

ErrorSingle[5](
	bAutoStatus:=AutoStatus,
	bResetPB:=PB_Reset,
	bBackLS:=LS_S1_Load_UpDownBack,
	bOutLS:=LS_S1_Load_UpDownOut,
	bSOL:=SOL_S1_Load_UpDown,
	bErrorStatus_Back=>Error_LS_S1_Load_UpDownBack,
	bErrorStatus_Out=>Error_LS_S1_Load_UpDownOut);

//異常
ErrorStatus_S1_Load:=
Error_LS_S1_Load_PanelUpDown1Back OR
Error_LS_S1_Load_PanelUpDown1Out OR
Error_LS_S1_Load_PanelUpDown2Back OR
Error_LS_S1_Load_PanelUpDown2Out OR
Error_LS_S1_Load_PanelClip1Back OR
Error_LS_S1_Load_PanelClip1Out OR
Error_LS_S1_Load_PanelClip2Back OR
Error_LS_S1_Load_PanelClip2Out;

ErrorStatus_S1_FeedPanelLoad:=
Error_LS_S1_Load_FixClipBack OR
Error_LS_S1_Load_FixClipOut OR
Error_LS_S1_Load_AlignmentClipBack OR
Error_LS_S1_Load_AlignmentClipOut OR
Error_LS_S1_Load_ConveyorClip1Back OR
Error_LS_S1_Load_ConveyorClip1Out OR
Error_LS_S1_Load_UpDownBack OR
Error_LS_S1_Load_UpDownOut;

//UNLOAD
ErrorDouble[2](
	bAutoStatus:=AutoStatus,
	bResetPB:=PB_Reset,
	bBackLS:=LS_S1_UnLoad_PanelUpDown1Back, bOutLS:=LS_S1_UnLoad_PanelUpDown1Out,
	bBackSOL:=SOL_S1_UnLoad_PanelUpDown1Back, bOutSOL:=SOL_S1_UnLoad_PanelUpDown1Out,
	bErrorStatus_Back=>Error_LS_S1_UnLoad_PanelUpDown1Back, bErrorStatus_Out=>Error_LS_S1_UnLoad_PanelUpDown1Out);

ErrorDouble[3](
	bAutoStatus:=AutoStatus,
	bResetPB:=PB_Reset,
	bBackLS:=LS_S1_UnLoad_PanelUpDown2Back, bOutLS:=LS_S1_UnLoad_PanelUpDown2Out,
	bBackSOL:=SOL_S1_UnLoad_PanelUpDown2Back,
	bOutSOL:=SOL_S1_UnLoad_PanelUpDown2Out,
	bErrorStatus_Back=>Error_LS_S1_UnLoad_PanelUpDown2Back,
	bErrorStatus_Out=>Error_LS_S1_UnLoad_PanelUpDown2Out);

ErrorSingle[6](
	bAutoStatus:=AutoStatus,
	bResetPB:=PB_Reset,
	bBackLS:=LS_S1_UnLoad_PanelClip1Back,
	bOutLS:=LS_S1_UnLoad_PanelClip1Out,
	bSOL:=SOL_S1_UnLoad_PanelClip,
	bErrorStatus_Back=>Error_LS_S1_UnLoad_PanelClip1Back,
	bErrorStatus_Out=>Error_LS_S1_UnLoad_PanelClip1Out);

ErrorSingle[7](
	bAutoStatus:=AutoStatus,
	bResetPB:=PB_Reset,
	bBackLS:=LS_S1_UnLoad_PanelClip2Back,
	bOutLS:=LS_S1_UnLoad_PanelClip2Out,
	bSOL:=SOL_S1_UnLoad_FixClip,
	bErrorStatus_Back=>Error_LS_S1_UnLoad_PanelClip2Back,
	bErrorStatus_Out=>Error_LS_S1_UnLoad_PanelClip2Out);

//UNLoad 後段
ErrorSingle[8](
	bAutoStatus:=AutoStatus,
	bResetPB:=PB_Reset,
	bBackLS:=LS_S1_UnLoad_FixClipBack,
	bOutLS:=LS_S1_UnLoad_FixClipOut,
	bSOL:=SOL_S1_UnLoad_FixClip,
	bErrorStatus_Back=>Error_LS_S1_UnLoad_FixClipBack,
	bErrorStatus_Out=>Error_LS_S1_UnLoad_FixClipOut);

ErrorSingle[9](
	bAutoStatus:=AutoStatus,
	bResetPB:=PB_Reset,
	bBackLS:=LS_S1_UnLoad_AlignmentClipBack,
	bOutLS:=LS_S1_UnLoad_AlignmentClipOut,
	bSOL:=SOL_S1_UnLoad_AlignmentClip,
	bErrorStatus_Back=>Error_LS_S1_UnLoad_AlignmentClipBack,
	bErrorStatus_Out=>Error_LS_S1_UnLoad_AlignmentClipOut);

ErrorSingle[10](
	bAutoStatus:=AutoStatus,
	bResetPB:=PB_Reset,
	bBackLS:=LS_S1_UnLoad_ConveyorClip1Back,
	bOutLS:=LS_S1_UnLoad_ConveyorClip1Out,
	bSOL:=SOL_S1_UnLoad_ConveyorClip,
	bErrorStatus_Back=>Error_LS_S1_UnLoad_ConveyorClip1Back,
	bErrorStatus_Out=>Error_LS_S1_UnLoad_ConveyorClip1Out);

ErrorSingle[11](
	bAutoStatus:=AutoStatus,
	bResetPB:=PB_Reset,
	bBackLS:=LS_S1_UnLoad_UpDownBack,
	bOutLS:=LS_S1_UnLoad_UpDownOut,
	bSOL:=SOL_S1_UnLoad_UpDown,
	bErrorStatus_Back=>Error_LS_S1_UnLoad_UpDownBack,
	bErrorStatus_Out=>Error_LS_S1_UnLoad_UpDownOut);
//異常
ErrorStatus_S1_UnLoad:=
Error_LS_S1_UnLoad_PanelUpDown1Back OR
Error_LS_S1_UnLoad_PanelUpDown1Out OR
Error_LS_S1_UnLoad_PanelUpDown2Back OR
Error_LS_S1_UnLoad_PanelUpDown2Out OR
Error_LS_S1_UnLoad_PanelClip1Back OR
Error_LS_S1_UnLoad_PanelClip1Out OR
Error_LS_S1_UnLoad_PanelClip2Back OR
Error_LS_S1_UnLoad_PanelClip2Out;

ErrorStatus_S1_FeedPanelUnLoad:=
Error_LS_S1_UnLoad_FixClipBack OR
Error_LS_S1_UnLoad_FixClipOut OR
Error_LS_S1_UnLoad_AlignmentClipBack OR
Error_LS_S1_UnLoad_AlignmentClipOut OR
Error_LS_S1_UnLoad_ConveyorClip1Back OR
Error_LS_S1_UnLoad_ConveyorClip1Out OR
Error_LS_S1_UnLoad_UpDownBack OR
Error_LS_S1_UnLoad_UpDownOut;

ErrorStatus_TH[1]:=
ErrorStatus_S1_Load OR
ErrorStatus_S1_UnLoad OR
ErrorStatus_S1_FeedPanelLoad OR
ErrorStatus_S1_FeedPanelUnLoad;

ErrorStatus[1]:=
YAMAHA_S_State_Alarm OR
YAMAHA_S_State_Warring OR
YAMAHA_Error_SOL_Clip;

ErrorStatus[16]:=
YAMAHA_S_State_Alarm OR
YAMAHA_S_State_Warring OR
YAMAHA_Error_SOL_Clip;
//**********************************************************************************************************************
(*機器停機異常*)
ErrorStatus_MachineStop:=
ErrorStatus[1] OR
ErrorStatus[2] OR
ErrorStatus[3] OR
ErrorStatus[4] OR
ErrorStatus[5] OR
ErrorStatus[6] OR
ErrorStatus[7] OR
ErrorStatus[8] OR
ErrorStatus[9] OR
ErrorStatus[10] OR 
ErrorStatus[11] OR
ErrorStatus[12] OR
ErrorStatus[13] OR
ErrorStatus[14] OR
ErrorStatus[15] OR
ErrorStatus[16] OR
ErrorStatus_TH[1] OR
ErrorStatus_TH[2] OR
ErrorStatus_TH[3] OR
ErrorStatus_TH[4] OR
ErrorStatus_TH[5] OR
ErrorStatus_TH[6] OR
ErrorStatus_TH[7] OR
ErrorStatus_TH[8] OR
ErrorStatus_TH[9] OR
ErrorStatus_TH[10] OR
ErrorStatus_TH[11] OR
ErrorStatus_TH[12] OR
ErrorStatus_TH[13] OR
ErrorStatus_TH[14] OR
ErrorStatus_TH[15] OR
ErrorStatus_TH[16];
(*機器不停機異常*)
ErrorStatus_MachineNonStop:=
Error_SNR_S1_Load_Full OR
Error_SNR_S1_UnLoad_Full OR
Error_SNR_S4_Load_Full OR
Error_SNR_S4_UnLoad_Full OR
Error_SNR_S6_Full OR
Error_SNR_S8_Full OR
Error_SNR_S10_Full;
(*異常排除*)
IF IndexData[17].ErrorLog[4]+
	IndexData[17].ErrorLog[5]+
	IndexData[17].ErrorLog[6]+
	IndexData[17].ErrorLog[7]+
	IndexData[17].ErrorLog[8]+
	IndexData[17].ErrorLog[9]+
	IndexData[17].ErrorLog[10]+
	IndexData[17].ErrorLog[11]+
	IndexData[17].ErrorLog[12]+
	IndexData[17].ErrorLog[13]+
	IndexData[17].ErrorLog[14]+
	IndexData[17].ErrorLog[15]+
	IndexData[17].ErrorLog[16]>0
	 THEN
	ErrorStatus_MachineStop_Record:=TRUE;
	ELSE
	ErrorStatus_MachineStop_Record:=FALSE;
END_IF;
//**********************************************************************************************************************
//異常RESET
IF PB_Reset THEN
	IndexData[17].ErrorLog[1]:=0;
	IndexData[17].ErrorLog[2]:=0;
	IndexData[17].ErrorLog[3]:=0;
	IndexData[17].ErrorLog[4]:=0;
	IndexData[17].ErrorLog[5]:=0;
	IndexData[17].ErrorLog[6]:=0;
	IndexData[17].ErrorLog[7]:=0;
	IndexData[17].ErrorLog[8]:=0;
	IndexData[17].ErrorLog[9]:=0;
	IndexData[17].ErrorLog[10]:=0;
	IndexData[17].ErrorLog[11]:=0;
	IndexData[17].ErrorLog[12]:=0;
	IndexData[17].ErrorLog[13]:=0;
	IndexData[17].ErrorLog[14]:=0;
	IndexData[17].ErrorLog[15]:=0;
	IndexData[17].ErrorLog[16]:=0;
END_IF;
END_PROGRAM

PROGRAM prStation1_PanelUnLoad
VAR
    Autoflow : INT;
    Initflow : INT;
    interlockback : ARRAY[0..2] OF BOOL;
    interlockout : ARRAY[0..2] OF BOOL;
    solStatus : ARRAY[0..2] OF BOOL;
    R_TRIG_1 : ARRAY[0..2] OF R_TRIG;
    F_TRIG_1 : F_TRIG;
    ErrorLS : BOOL;
    StartFlag : BOOL;
    TON_1 : TON;
END_VAR
VAR_EXTERNAL
    RY_S1_UnLoad_VariableSpeedMotor : BOOL;
    HMIPB_SOL_S1_UnLoad_PanelUpDown1Back : BOOL;
    AutoStatus : BOOL;
    SOL_S1_UnLoad_PanelUpDown1Back : BOOL;
    SOL_S1_UnLoad_PanelUpDown1Out : BOOL;
    LS_S1_UnLoad_PanelUpDown1Back : BOOL;
    HMIPB_SOL_S1_UnLoad_PanelUpDown1Out : BOOL;
    LS_S1_UnLoad_PanelUpDown1Out : BOOL;
    HMIPB_SOL_S1_UnLoad_PanelUpDown2Back : BOOL;
    SOL_S1_UnLoad_PanelUpDown2Back : BOOL;
    SOL_S1_UnLoad_PanelUpDown2Out : BOOL;
    LS_S1_UnLoad_PanelUpDown2Back : BOOL;
    HMIPB_SOL_S1_UnLoad_PanelUpDown2Out : BOOL;
    LS_S1_UnLoad_PanelUpDown2Out : BOOL;
    HMIPB_SOL_S1_UnLoad_PanelClip : BOOL;
    SOL_S1_UnLoad_PanelClip : BOOL;
    ErrorStatus_S1_UnLoad : BOOL;
    SNR_S1_UnLoad_PanelFeed : BOOL;
    SystemReadyStatus : BOOL;
    Error_PB_EStop : BOOL;
    LS_S1_UnLoad_PanelClip1Out : BOOL;
    LS_S1_UnLoad_PanelClip2Out : BOOL;
    LS_S1_UnLoad_PanelClip1Back : BOOL;
    LS_S1_UnLoad_PanelClip2Back : BOOL;
END_VAR
(*
程序名稱: Panel UNLOAD程序
作者:蔡相偉
版本,日期,版本資訊:
1.0.0		2017/11/16		初始版本

PowerOn=0
Idle=1
Panel出盤程序開始=10
第1段出=2
夾持出=3
第2段出=4
夾持回=5
第1段,第2段回=6
*)
//***************************************************************************************************************
//Define
ErrorLS:=ErrorStatus_S1_UnLoad;
StartFlag:=TON_1.Q;
TON_1(In:=(SNR_S1_UnLoad_PanelFeed) AND NOT(RY_S1_UnLoad_VariableSpeedMotor), PT:=t#5s);
//PowerOn=0
IF NOT(SystemReadyStatus AND NOT(ErrorLS) AND  NOT(Error_PB_EStop) AND AutoStatus) THEN
	Autoflow:=0;
END_IF;

//Idle=1
IF AutoFlow=0 AND SystemReadyStatus AND NOT(ErrorLS) AND  NOT(Error_PB_Estop) AND AutoStatus THEN
	AutoFlow:=1;
END_IF;

IF Autoflow=6 AND LS_S1_UnLoad_PanelUpDown1Back AND LS_S1_UnLoad_PanelUpDown2Back THEN
	Autoflow:=1;
END_IF;

//第1段出=2
IF Autoflow=1 AND StartFlag THEN
	Autoflow:=2;
END_IF;

//承盤夾持出=3
IF Autoflow=2 AND LS_S1_UnLoad_PanelUpDown1Out THEN
	Autoflow:=3;
END_IF;

//第2段出=4
IF Autoflow=3 AND LS_S1_UnLoad_PanelClip1Out AND LS_S1_UnLoad_PanelClip2Out THEN
	Autoflow:=4;
END_IF;

//承盤夾持回=5
IF Autoflow=4 AND LS_S1_UnLoad_PanelUpDown2Out THEN
	Autoflow:=5;
END_IF;

//第1段,第2段回=6
IF Autoflow=5 AND  LS_S1_UnLoad_PanelClip1Back AND LS_S1_UnLoad_PanelClip2Back THEN
	Autoflow:=6;
END_IF;

//***************************************************************************************************************
//下夾板出盤下降第1段回電磁閥
interlockback[0]:=NOT(RY_S1_UnLoad_VariableSpeedMotor);
IF ((HMIPB_SOL_S1_UnLoad_PanelUpDown1Back AND NOT(AutoStatus)) OR Autoflow=6 OR Initflow=6) AND interlockback[0] THEN
	SOL_S1_UnLoad_PanelUpDown1Back:=TRUE;
	SOL_S1_UnLoad_PanelUpDown1Out:=FALSE;
END_IF;
IF LS_S1_UnLoad_PanelUpDown1Back THEN
	SOL_S1_UnLoad_PanelUpDown1Back:=FALSE;
END_IF;

//下夾板出盤下降第1段出電磁閥
interlockout[0]:=TRUE;
IF ((HMIPB_SOL_S1_UnLoad_PanelUpDown1Out AND NOT(AutoStatus)) OR Autoflow=2) AND interlockout[0] THEN
	SOL_S1_UnLoad_PanelUpDown1Back:=FALSE;
	SOL_S1_UnLoad_PanelUpDown1Out:=TRUE;
END_IF;
IF LS_S1_UnLoad_PanelUpDown1Out THEN
	SOL_S1_UnLoad_PanelUpDown1Out:=FALSE;
END_IF;
//***************************************************************************************************************
//下夾板出盤下降第2段回電磁閥
interlockback[1]:=TRUE;
IF ((HMIPB_SOL_S1_UnLoad_PanelUpDown2Back AND NOT(AutoStatus)) OR Autoflow=6 OR Initflow=6) AND interlockback[1] THEN
	SOL_S1_UnLoad_PanelUpDown2Back:=TRUE;
	SOL_S1_UnLoad_PanelUpDown2Out:=FALSE;
END_IF;
IF LS_S1_UnLoad_PanelUpDown2Back THEN
	SOL_S1_UnLoad_PanelUpDown2Back:=FALSE;
END_IF;

//下夾板出盤下降第2段出電磁閥
interlockout[1]:=LS_S1_UnLoad_PanelClip1Out AND LS_S1_UnLoad_PanelClip2Out AND SOL_S1_UnLoad_PanelClip;
IF ((HMIPB_SOL_S1_UnLoad_PanelUpDown2Out AND NOT(AutoStatus)) OR Autoflow=4) AND interlockout[1] THEN
	SOL_S1_UnLoad_PanelUpDown2Back:=FALSE;
	SOL_S1_UnLoad_PanelUpDown2Out:=TRUE;
END_IF;
IF LS_S1_UnLoad_PanelUpDown2Out THEN
	SOL_S1_UnLoad_PanelUpDown2Out:=FALSE;
END_IF;
//***************************************************************************************************************
(*下夾板出盤承載電磁閥*)
R_TRIG_1[2](CLK:=HMIPB_SOL_S1_UnLoad_PanelClip AND NOT(AutoStatus));
interlockback[2]:=TRUE;
interlockout[2]:=LS_S1_UnLoad_PanelUpDown1Out;
(*SET*)
IF ((R_TRIG_1[2].Q AND NOT(solStatus[2])) OR Autoflow=3) AND interlockout[2] THEN
	SOL_S1_UnLoad_PanelClip:=TRUE;
END_IF;
(*RESET*)
IF ((R_TRIG_1[2].Q AND (solStatus[2])) OR Autoflow=5 OR Initflow=5) AND interlockback[2] THEN
	SOL_S1_UnLoad_PanelClip:=FALSE;
END_IF;
(*STATUS*)
solStatus[2]:=SOL_S1_UnLoad_PanelClip;

//***************************************************************************************************************
(*
程序名稱: Panel LOAD RESET程序
作者:蔡相偉
版本,日期,版本資訊:
1.0.0		2017/11/16		初始版本

PowerOn=0
Idle=1
第2段回=4
夾持回=5
第1段回=6

//***************************************************************************************************************
//PowerOn=0
IF NOT(SystemReadyStatus) THEN
	Initflow:=0;
END_IF;

//Idle=1
IF Initflow=0 AND SystemReadyStatus THEN
	Initflow:=1;
END_IF;

IF Initflow=6 AND LS_S1_Load_PanelUpDown1Back THEN
	Initflow:=1;
END_IF;

F_TRIG_1(Clk:=ErrorLS);
//第2段回=4
IF Initflow=1 AND F_TRIG_1.Q THEN
	Initflow:=4;
END_IF;

//承盤夾持回=5
IF Initflow=4 AND LS_S1_Load_PanelUpDown2Back THEN
	Initflow:=5;
END_IF;

//第1段回=6
IF Initflow=5 AND  LS_S1_Load_PanelClip1Back AND LS_S1_Load_PanelClip2Back THEN
	Initflow:=6;
END_IF;
*)
END_PROGRAM

PROGRAM prStation1_FeedPanelUnLoad
VAR
    Autoflow : INT;
    interlockback : ARRAY[0..3] OF BOOL;
    interlockout : ARRAY[0..3] OF BOOL;
    solStatus : ARRAY[0..3] OF BOOL;
    R_TRIG_1 : ARRAY[0..3] OF R_TRIG;
    ErrorLS : BOOL;
    StartFlag : BOOL;
    TON_1 : TON;
    TON_2 : TON;
    TON_3 : TON;
    TON_4 : TON;
    TON_5 : TON;
    TON_6 : TON;
    TON_7 : TON;
    F_TRIG_1 : F_TRIG;
END_VAR
VAR_EXTERNAL
    HMIPB_SOL_S1_UnLoad_FixClip : BOOL;
    SOL_S1_UnLoad_FixClip : BOOL;
    AutoStatus : BOOL;
    HMIPB_SOL_S1_UnLoad_AlignmentClip : BOOL;
    SOL_S1_UnLoad_AlignmentClip : BOOL;
    HMIPB_SOL_S1_UnLoad_ConveyorClip : BOOL;
    SOL_S1_UnLoad_ConveyorClip : BOOL;
    HMIPB_SOL_S1_UnLoad_UpDown : BOOL;
    SOL_S1_UnLoad_UpDown : BOOL;
    SNR_S1_UnLoad_PanelFeed : BOOL;
    HMIPB_RY_S1_UnLoad_VariableSpeedMotor : BOOL;
    RY_S1_UnLoad_VariableSpeedMotor : BOOL;
    SNR_S1_UnLoad_PanelClip : BOOL;
    HMIPB_RY_S1_UnLoad_FixSpeedMotor : BOOL;
    RY_S1_UnLoad_FixSpeedMotor : BOOL;
    ErrorStatus_S1_FeedPanelUnLoad : BOOL;
    SystemReadyStatus : BOOL;
    Error_PB_EStop : BOOL;
    YAMAHA_Unload_ChangePanelStart : BOOL;
    HMIPB_YAMAHA_Unload_ChangePanelStart : BOOL;
    YAMAHA_Load_Ready : BOOL;
    YAMAHA_UnLoad_Ready : BOOL;
    LS_S1_UnLoad_AlignmentClipBack : BOOL;
    YAMAHA_Unload_OKStart : BOOL;
    LS_S1_UnLoad_FixClipOut : BOOL;
    LS_S1_UnLoad_AlignmentClipOut : BOOL;
    LS_S1_UnLoad_ConveyorClip1Out : BOOL;
    LS_S1_UnLoad_ConveyorClip2Out : BOOL;
    SNR_S1_Load_Feed : BOOL;
    HMIPB_RY_S1_Center_VariableSpeedMotor : BOOL;
    RY_S1_Center_VariableSpeedMotor : BOOL;
    SNR_S1_UnLoad_Feed : BOOL;
    LS_S1_UnLoad_UpDownOut : BOOL;
    LS_S1_UnLoad_ConveyorClip1Back : BOOL;
    LS_S1_UnLoad_ConveyorClip2Back : BOOL;
    LS_S1_UnLoad_UpDownBack : BOOL;
    LS_S1_UnLoad_FixClipBack : BOOL;
END_VAR
(*
程序名稱: 收盤程序
作者:蔡相偉
版本,日期,版本資訊:
1.0.0		2017/11/16		初始版本

PowerOn=0--->
Idle=1--->
換盤程序開始=2|--->工件取放處無盤=10--->固定,活動,軌道夾持出=11--->上下出=12--->軌道夾持回=13--->上下回=14--->固定夾持回=15--->活動夾持回=16--->換盤完成=17--->1
						  |--->工件取放處有盤=20--->軌道夾持回=21--->固定,活動夾持出=22--->馬達ON=23--->馬達運行中=24--->盤離位,定速馬達停止=25--->10
*)
(*
Error Code
1:緊急停止
2:磁簧異常
*)
//***************************************************************************************************************
//Define
ErrorLS:=
ErrorStatus_S1_FeedPanelUnLoad;
//***************************************************************************************************************
//PowerOn=0
IF NOT(SystemReadyStatus AND NOT(ErrorLS) AND  NOT(Error_PB_EStop) AND AutoStatus) THEN
	Autoflow:=0;
END_IF;

//Idle=1
IF Autoflow=0 AND SystemReadyStatus AND NOT(ErrorLS) AND  NOT(Error_PB_Estop) AND AutoStatus THEN
	Autoflow:=1;
END_IF;

IF Autoflow=17 AND NOT(YAMAHA_Unload_ChangePanelStart) THEN
	Autoflow:=1;
END_IF;

TON_1(In:=Autoflow=1 AND NOT(SNR_S1_UnLoad_PanelClip), PT:=t#1s);

TON_7(In:=(SNR_S1_UnLoad_PanelClip), PT:=t#1s);
IF Autoflow=1 AND TON_7.Q THEN		(*READY訊號*)
	YAMAHA_UnLoad_Ready:=TRUE;
ELSE
	YAMAHA_UnLoad_Ready:=FALSE;
END_IF;
//換盤程序開始=2
IF Autoflow=1 AND (YAMAHA_Unload_ChangePanelStart OR HMIPB_YAMAHA_Unload_ChangePanelStart OR TON_1.Q) THEN
	Autoflow:=2;
END_IF;
IF Autoflow=2 THEN
	HMIPB_RY_S1_Center_VariableSpeedMotor:=TRUE;
END_IF;

//工件取放處無盤=10
IF Autoflow=2 AND (RY_S1_Center_VariableSpeedMotor OR SNR_S1_UnLoad_Feed) AND NOT(SNR_S1_UnLoad_PanelClip) THEN
	Autoflow:=10;
END_IF;

IF Autoflow=25 THEN
	Autoflow:=10;
END_IF;

//固定,活動,軌道夾持出=11
IF Autoflow=10 THEN
	Autoflow:=11;
END_IF;
TON_4(In:=(SNR_S1_UnLoad_Feed), PT:=t#1s);
//上下出=12
IF Autoflow=11 AND LS_S1_UnLoad_FixClipOut AND LS_S1_UnLoad_AlignmentClipOut AND LS_S1_UnLoad_ConveyorClip1Out AND LS_S1_UnLoad_ConveyorClip2Out AND TON_4.Q THEN
	Autoflow:=12;
END_IF;

//軌道夾持回=13
IF Autoflow=12 AND LS_S1_UnLoad_UpDownOut THEN
	Autoflow:=13;
END_IF;

//上下回=14
IF Autoflow=13 AND LS_S1_UnLoad_ConveyorClip1Back AND LS_S1_UnLoad_ConveyorClip2Back THEN
	Autoflow:=14;
END_IF;

//固定夾持回=15
IF Autoflow=14 AND LS_S1_UnLoad_UpDownBack THEN
	Autoflow:=15;
END_IF;

//活動夾持回=16
IF Autoflow=15 AND LS_S1_UnLoad_FixClipBack THEN
	Autoflow:=16;
END_IF;

//換盤完成=17
IF Autoflow=16 AND LS_S1_UnLoad_AlignmentClipBack THEN
	Autoflow:=17;
END_IF;

//***************************************************************************************************************
//工件取放處有盤=20
IF Autoflow=2 AND (RY_S1_Center_VariableSpeedMotor OR SNR_S1_UnLoad_Feed) AND (SNR_S1_UnLoad_PanelClip) THEN
	Autoflow:=20;
END_IF;

//軌道夾持回=21
IF Autoflow=20 THEN
	Autoflow:=21;
END_IF;

//固定,活動夾持出=22
IF Autoflow=21 AND LS_S1_UnLoad_ConveyorClip1Back AND LS_S1_UnLoad_ConveyorClip2Back THEN
	Autoflow:=22;
END_IF;

//馬達ON=23
IF Autoflow=22 AND LS_S1_UnLoad_FixClipOut AND LS_S1_UnLoad_AlignmentClipOut AND NOT(SNR_S1_UnLoad_PanelFeed) THEN
	Autoflow:=23;
END_IF;
IF Autoflow=23 THEN
	HMIPB_RY_S1_UnLoad_FixSpeedMotor:=TRUE;
	HMIPB_RY_S1_UnLoad_VariableSpeedMotor:=TRUE;
END_IF;

//馬達運行中=24
IF Autoflow=23 AND RY_S1_UnLoad_FixSpeedMotor AND RY_S1_UnLoad_VariableSpeedMotor THEN
	Autoflow:=24;
END_IF;

//盤離位,定速馬達停止=25
IF Autoflow=24 AND NOT(SNR_S1_UnLoad_PanelClip) AND NOT(RY_S1_UnLoad_FixSpeedMotor) THEN
	Autoflow:=25;
END_IF;

//***************************************************************************************************************
//下夾板出盤固定邊定位電磁閥
R_TRIG_1[0](CLK:=HMIPB_SOL_S1_UnLoad_FixClip AND NOT(AutoStatus));
interlockback[0]:=TRUE;
interlockout[0]:=TRUE;
//SET
IF ((R_TRIG_1[0].Q AND NOT(solStatus[0])) OR Autoflow=11 OR Autoflow=22) AND interlockout[0] THEN
	SOL_S1_UnLoad_FixClip:=TRUE;
END_IF;
//RESET
IF ((R_TRIG_1[0].Q AND (solStatus[0])) OR Autoflow=15) AND interlockback[0] THEN
	SOL_S1_UnLoad_FixClip:=FALSE;
END_IF;
//STATUS
solStatus[0]:=SOL_S1_UnLoad_FixClip;
//***************************************************************************************************************
//下夾板出盤活動邊定位電磁閥
R_TRIG_1[1](CLK:=HMIPB_SOL_S1_UnLoad_AlignmentClip AND NOT(AutoStatus));
interlockback[1]:=TRUE;
interlockout[1]:=TRUE;
//SET
IF ((R_TRIG_1[1].Q AND NOT(solStatus[1])) OR Autoflow=11 OR Autoflow=22) AND interlockout[1] THEN
	SOL_S1_UnLoad_AlignmentClip:=TRUE;
END_IF;
//RESET
IF ((R_TRIG_1[1].Q AND (solStatus[1])) OR Autoflow=16) AND interlockback[1] THEN
	SOL_S1_UnLoad_AlignmentClip:=FALSE;
END_IF;
//STATUS
solStatus[1]:=SOL_S1_UnLoad_AlignmentClip;
//***************************************************************************************************************
//下夾板出盤軌道開合電磁閥
R_TRIG_1[2](CLK:=HMIPB_SOL_S1_UnLoad_ConveyorClip AND NOT(AutoStatus));
interlockback[2]:=TRUE;
interlockout[2]:=TRUE;
//SET
IF ((R_TRIG_1[2].Q AND NOT(solStatus[2])) OR Autoflow=11) AND interlockout[2] THEN
	SOL_S1_UnLoad_ConveyorClip:=TRUE;
END_IF;
//RESET
IF ((R_TRIG_1[2].Q AND (solStatus[2])) OR Autoflow=13 OR Autoflow=21) AND interlockback[2] THEN
	SOL_S1_UnLoad_ConveyorClip:=FALSE;
END_IF;
//STATUS
solStatus[2]:=SOL_S1_UnLoad_ConveyorClip;
//***************************************************************************************************************
//下夾板出盤升降電磁閥
R_TRIG_1[3](CLK:=HMIPB_SOL_S1_UnLoad_UpDown AND NOT(AutoStatus));
interlockback[3]:=TRUE;
interlockout[3]:=LS_S1_UnLoad_ConveyorClip1Out AND LS_S1_UnLoad_ConveyorClip2Out AND SOL_S1_UnLoad_ConveyorClip;
//SET
IF ((R_TRIG_1[3].Q AND NOT(solStatus[3])) OR Autoflow=12) AND interlockout[3] THEN
	SOL_S1_UnLoad_UpDown:=TRUE;
END_IF;
//RESET
IF ((R_TRIG_1[3].Q AND (solStatus[3])) OR Autoflow=14) AND interlockback[3] THEN
	SOL_S1_UnLoad_UpDown:=FALSE;
END_IF;
//STATUS
solStatus[3]:=SOL_S1_UnLoad_UpDown;
//***************************************************************************************************************
//下夾板出盤調速馬達繼電器
//RESET
TON_6(In:=(SNR_S1_UnLoad_PanelFeed), PT:=t#1s);
IF TON_6.Q THEN
	HMIPB_RY_S1_UnLoad_VariableSpeedMotor:=FALSE;
END_IF;
//OUT
RY_S1_UnLoad_VariableSpeedMotor:=HMIPB_RY_S1_UnLoad_VariableSpeedMotor;
//***************************************************************************************************************
//下夾板出盤定速馬達繼電器
//RESET
TON_5(In:=NOT(SNR_S1_UnLoad_PanelClip), PT:=t#1s);
IF TON_5.Q THEN
	HMIPB_RY_S1_UnLoad_FixSpeedMotor:=FALSE;
END_IF;
//OUT
RY_S1_UnLoad_FixSpeedMotor:=HMIPB_RY_S1_UnLoad_FixSpeedMotor;
END_PROGRAM

PROGRAM prSystemInit
VAR
    SystemInitFlow : INT := 0;
    TON1 : TON;
    TON_3 : TON;
    R_TRIG_3 : R_TRIG;
END_VAR
VAR_EXTERNAL
    AutoStatus : BOOL;
    SystemReadyStatus : BOOL;
    PB_EStop : BOOL;
    Error_PB_EStop : BOOL;
    Manual2AutoFlag : BOOL;
    ErrorStatus_MachineStop : BOOL;
    ErrorStatus_MachineNonStop : BOOL;
    ErrorStatus_MachineStop_Record : BOOL;
    BZ : BOOL;
    RL : BOOL;
    GL : BOOL;
    YL : BOOL;
END_VAR
(******************************************************************
程式:系統初始化
作者:蔡相偉
版本資訊:1.0.0		2016/5/26

全部狀態RESET=0
伺服上電=1
伺服未回HOME=2
伺服Servo on=3
伺服Ready=4
夾爪回=5
夾爪前後回=6
伺服上下軸Serch Home=7
伺服上下軸Serch Home中=8
伺服上下軸Serch Home完成=9
伺服橫移軸Serch Home=10
伺服橫移軸Serch Home中=11
伺服橫移軸Serch Home完成=12
自動SET=13
系統READY SET=14
Init完成=15
******************************************************************)
//全部狀態RESET=0
IF P_First_Run THEN
	SystemInitFlow:=0;
	AutoStatus:=FALSE;
	SystemReadyStatus:=FALSE;
END_IF;

//伺服上電=1
IF SystemInitFlow=0 AND P_Off AND PB_EStop AND NOT(Error_PB_EStop) AND NOT(AutoStatus) AND NOT(SystemReadyStatus) (*AND MC_Axis000.DrvStatus.MainPower AND MC_Axis001.DrvStatus.MainPower*) THEN
	SystemInitFlow:=1;
END_IF;

//伺服未回HOME=2
IF SystemInitFlow=1 (*AND (NOT(MC_Axis000.Details.Homed) OR NOT(MC_Axis001.Details.Homed))*) THEN
	SystemInitFlow:=2;
END_IF;

//伺服Servo on=3
IF SystemInitFlow=2 THEN
	SystemInitFlow:=3;
END_IF;
IF SystemInitFlow=3 THEN
	//PB_ServoOn_UpDown:=TRUE;
	//PB_ServoOn_Move:=TRUE;
	;
END_IF;

//伺服Ready=4
IF SystemInitFlow=3 (*AND AxMove.bServoOn AND AxUpDown.bServoOn AND MC_Axis000.DrvStatus.Ready AND MC_Axis001.DrvStatus.Ready*) THEN
	SystemInitFlow:=4;
END_IF;

//夾爪回=5
TON1(In:=SystemInitFlow=4 , PT:=t#1s);
IF SystemInitFlow=4 AND TON1.Q THEN
	SystemInitFlow:=5;
END_IF;
IF SystemInitFlow=5 THEN
	;
END_IF;

//夾爪前後回=6
IF SystemInitFlow=5 THEN
	SystemInitFlow:=6;
END_IF;
IF SystemInitFlow=6 THEN
	//SOL_Move:=FALSE;
	;
END_IF;

//伺服上下軸Serch Home=7
IF SystemInitFlow=6  THEN
	SystemInitFlow:=7;
END_IF;
IF SystemInitFlow=7 THEN
	//AxUpDown.pbSerchHome:=TRUE;
	;
END_IF;

//伺服上下軸Serch Home中=8
IF SystemInitFlow=7 THEN
	//AxUpDown.pbSerchHome:=FALSE;
	SystemInitFlow:=8;
END_IF;

//伺服上下軸Serch Home完成=9
IF SystemInitFlow=8  THEN
	SystemInitFlow:=9;
END_IF;

//伺服橫移軸Serch Home=10
IF SystemInitFlow=9  THEN
	SystemInitFlow:=10;
END_IF;
IF SystemInitFlow=10 THEN
	//AxMove.pbSerchHome:=TRUE;
	;
END_IF;

//伺服橫移軸Serch Home中=11
IF SystemInitFlow=10 THEN
	//AxMove.pbSerchHome:=FALSE;
	SystemInitFlow:=11;
END_IF;

//伺服橫移軸Serch Home完成=12
IF SystemInitFlow=11 THEN
	SystemInitFlow:=12;
END_IF;

//自動SET=13
IF SystemInitFlow=12  THEN
	SystemInitFlow:=13;
END_IF;
IF SystemInitFlow=13 THEN
	AutoStatus:=TRUE;
END_IF;

//系統READY SET=14
IF SystemInitFlow=13 AND AutoStatus THEN
	SystemInitFlow:=14;
END_IF;
IF SystemInitFlow=14 THEN
	SystemReadyStatus:=TRUE;
END_IF;

//Init完成=15
IF SystemInitFlow=14 AND SystemReadyStatus THEN
	SystemInitFlow:=15;
END_IF;

//******************************************************************
//手動轉自動
R_TRIG_3(CLK:= AutoStatus ,Q=> Manual2AutoFlag );

(******************************************************************
程式:燈號及蜂鳴器
作者:蔡相偉
版本資訊:1.0.0		2016/5/26
******************************************************************)
//BZ停止
TON_3(IN:=(ErrorStatus_MachineStop OR ErrorStatus_MachineNonStop OR ErrorStatus_MachineStop_Record) , PT:=t#10s);
//BZ
IF (ErrorStatus_MachineStop OR ErrorStatus_MachineNonStop OR ErrorStatus_MachineStop_Record) AND NOT(TON_3.Q) THEN
	BZ:=TRUE;
	ELSE
	BZ:=FALSE;
END_IF;
//紅燈
IF ErrorStatus_MachineStop OR ErrorStatus_MachineStop_Record THEN
	RL:=TRUE;
	ELSE
	RL:=FALSE;
END_IF;
//綠燈
IF NOT(ErrorStatus_MachineStop) AND
	NOT(ErrorStatus_MachineNonStop) AND NOT(ErrorStatus_MachineStop_Record) THEN
	GL:=TRUE;
	ELSE
	GL:=FALSE;
END_IF;
//黃燈
IF ErrorStatus_MachineNonStop THEN
	YL:=TRUE;
	ELSE
	YL:=FALSE;
END_IF;
END_PROGRAM

PROGRAM prStation1
VAR
    AutoFlow : INT;
    Rtrig_test : R_TRIG;
END_VAR
VAR_EXTERNAL
    IndexData : ARRAY[0..19] OF stIndexData;
    DisablePB : ARRAY[0..19] OF BOOL;
    TestPB : ARRAY[0..19] OF BOOL;
    SystemReadyStatus : BOOL;
    ErrorStatus : ARRAY[0..19] OF BOOL;
    Error_PB_EStop : BOOL;
    AutoStatus : BOOL;
    MachineRunStatus : BOOL;
    YAMAHA_Load_Start : BOOL;
    YAMAHA_Load_Finish : BOOL;
    YAMAHA_Error_SOL_Clip : BOOL;
END_VAR
(*
程序名稱:第1站上料流程
作者:蔡相偉
版本,日期,版本資訊:
1.0.0		2017/11/21		初始版本
PowerOn=0
Idle=1
上料開始=2
上料完成=3
*)
//本站狀態判斷
IF IndexData[1].OKFlag[1]
	OR IndexData[1].NGFlag[1] THEN
	IndexData[1].FinishFlag[1]:=TRUE;
END_IF;
(*
//前站狀態判斷
IF NOT(IndexData[10].FinishFlag[9]
	AND IndexData[10].OKFlag[9]
	AND NOT(IndexData[10].NGFlag[9])) THEN
	IndexData[10].NGFlag[10]:=TRUE;
END_IF;
*)
//本站關閉判斷
IF DisablePB[1] THEN
	IndexData[1].NGFlag[1]:=TRUE;
END_IF;

Rtrig_test(CLK:=TestPB[1]);
//PowerOn=0
IF NOT(SystemReadyStatus AND AutoStatus AND NOT(ErrorStatus[1]) AND NOT(Error_PB_EStop)) THEN
	Autoflow:=0;
END_IF;

//Idle=1
IF AutoFlow=0 AND SystemReadyStatus AND AutoStatus AND NOT(ErrorStatus[1]) AND NOT(Error_PB_EStop) THEN
	AutoFlow:=1;
END_IF;

IF AutoFlow=3 AND NOT(YAMAHA_Load_Start) AND IndexData[1].FinishFlag[1] THEN
	AutoFlow:=1;
END_IF;

//上料開始=2
IF Autoflow=1
	AND AutoStatus
	AND NOT(DisablePB[1])
	AND (MachineRunStatus AND NOT(IndexData[1].FinishFlag[1]) OR Rtrig_test.Q) THEN
	Autoflow:=2;
END_IF;
IF AutoFlow=2 THEN
	YAMAHA_Load_Start:=TRUE;
END_IF;
IF YAMAHA_Load_Finish OR AutoFlow=0 THEN
	YAMAHA_Load_Start:=FALSE;
END_IF;

//上料完成=3
IF AutoFlow=2 AND (YAMAHA_Load_Finish) THEN
	AutoFlow:=3;
END_IF;
IF AutoFlow=3 THEN
	IndexData[1].OKFlag[1]:=TRUE;
END_IF;
END_PROGRAM

PROGRAM prStation16
VAR
    AutoFlow : INT;
    Rtrig_test : R_TRIG;
    Rtrig_test2 : R_TRIG;
END_VAR
VAR_EXTERNAL
    IndexData : ARRAY[0..19] OF stIndexData;
    DisablePB : ARRAY[0..19] OF BOOL;
    TestPB : ARRAY[0..19] OF BOOL;
    SystemReadyStatus : BOOL;
    ErrorStatus : ARRAY[0..19] OF BOOL;
    Error_PB_EStop : BOOL;
    AutoStatus : BOOL;
    MachineRunStatus : BOOL;
    HMIPB_YAMAHA_Unload_OKStart : BOOL;
    YAMAHA_Unload_OKStart : BOOL;
    YAMAHA_Unload_Finish : BOOL;
    HMIPB_YAMAHA_Unload_NGStart : BOOL;
    YAMAHA_Unload_NGStart : BOOL;
END_VAR
(*
程序名稱:第16站下料流程
作者:蔡相偉
版本,日期,版本資訊:
1.0.0		2017/11/21		初始版本
PowerOn=0
Idle=1|--->OK下料開始=10--->OK下料完成=11
		  |--->NG下料開始=20--->NG下料完成=21
*)
//本站狀態判斷
IF IndexData[16].OKFlag[16]
	OR IndexData[16].NGFlag[16] THEN
	IndexData[16].FinishFlag[16]:=TRUE;
END_IF;

//前站狀態判斷
IF NOT(IndexData[16].OKFlag[1]) THEN
	IndexData[16].NGFlag[16]:=TRUE;
END_IF;

(*
//本站關閉判斷
IF DisablePB[1] THEN
	IndexData[1].NGFlag[1]:=TRUE;
END_IF;
*)
Rtrig_test(CLK:=HMIPB_YAMAHA_Unload_OKStart);
Rtrig_test2(CLK:=HMIPB_YAMAHA_Unload_NGStart);
//PowerOn=0
IF NOT(SystemReadyStatus AND AutoStatus AND NOT(ErrorStatus[16]) AND NOT(Error_PB_EStop)) THEN
	Autoflow:=0;
END_IF;

//Idle=1
IF AutoFlow=0 AND SystemReadyStatus AND AutoStatus AND NOT(ErrorStatus[16]) AND NOT(Error_PB_EStop) THEN
	AutoFlow:=1;
END_IF;

IF AutoFlow=11 AND NOT(YAMAHA_Unload_OKStart) AND IndexData[16].FinishFlag[16] THEN
	AutoFlow:=1;
END_IF;

IF AutoFlow=21 AND NOT(YAMAHA_Unload_NGStart) AND IndexData[16].FinishFlag[16] THEN
	AutoFlow:=1;
END_IF;

//OK下料開始=10
IF Autoflow=1
	AND AutoStatus
	AND NOT(DisablePB[16])
	AND (MachineRunStatus AND NOT(IndexData[16].FinishFlag[16]) AND IndexData[16].OKFlag[1] AND IndexData[16].FinishFlag[15] AND IndexData[16].OKFlag[15] AND NOT(IndexData[16].NGFlag[15]) OR Rtrig_test.Q) THEN
	Autoflow:=10;
END_IF;
IF AutoFlow=10 THEN
	YAMAHA_Unload_OKStart:=TRUE;
END_IF;
IF YAMAHA_Unload_Finish OR AutoFlow=0 THEN
	YAMAHA_Unload_OKStart:=FALSE;
END_IF;

//OK下料完成=11
IF AutoFlow=10 AND (YAMAHA_Unload_Finish) THEN
	AutoFlow:=11;
END_IF;
IF AutoFlow=11 THEN
	IndexData[16].OKFlag[16]:=TRUE;
END_IF;

//NG下料開始=20
IF Autoflow=1
	AND AutoStatus
	AND NOT(DisablePB[16])
	AND (MachineRunStatus AND NOT(IndexData[16].FinishFlag[16]) AND IndexData[16].OKFlag[1] AND IndexData[16].FinishFlag[15] AND (IndexData[16].NGFlag[15]) OR Rtrig_test2.Q) THEN
	Autoflow:=20;
END_IF;
IF AutoFlow=20 THEN
	YAMAHA_Unload_NGStart:=TRUE;
END_IF;
IF YAMAHA_Unload_Finish OR AutoFlow=0 THEN
	YAMAHA_Unload_NGStart:=FALSE;
END_IF;

//NG下料完成=21
IF AutoFlow=20 AND (YAMAHA_Unload_Finish) THEN
	AutoFlow:=21;
END_IF;
IF AutoFlow=21 THEN
	IndexData[16].NGFlag[16]:=TRUE;
END_IF;
END_PROGRAM

PROGRAM prStation4
VAR
    interlockback : ARRAY[0..3] OF BOOL;
    interlockout : ARRAY[0..3] OF BOOL;
    solstatus : ARRAY[0..3] OF BOOL;
    R_TRIG_1 : ARRAY[0..3] OF R_TRIG;
    Rtrig_test : R_TRIG;
    F_TRIG_1 : F_TRIG;
    Autoflow : INT;
    Initflow : INT;
    TON1 : TON;
    TON2 : TON;
END_VAR
VAR_EXTERNAL
    HMIPB_SOL_S4_MoveBack : BOOL;
    AutoStatus : BOOL;
    SOL_S4_MoveBack : BOOL;
    SOL_S4_MoveOut : BOOL;
    LS_S4_MoveBack : BOOL;
    HMIPB_SOL_S4_MoveOut : BOOL;
    LS_S4_MoveOut : BOOL;
    HMIPB_SOL_S4_UpDown : BOOL;
    SOL_S4_UpDown : BOOL;
    HMIPB_SOL_S4_Clip : BOOL;
    SOL_S4_Clip : BOOL;
    IndexData : ARRAY[0..19] OF stIndexData;
    DisablePB : ARRAY[0..19] OF BOOL;
    TestPB : ARRAY[0..19] OF BOOL;
    SystemReadyStatus : BOOL;
    ErrorStatus : ARRAY[0..19] OF BOOL;
    Error_PB_EStop : BOOL;
    SOL_S4_THMoveBack : BOOL;
    Error_SNR_S4_Feed : BOOL;
    LS_S4_THMoveBack : BOOL;
    LS_S4_UpDownBack : BOOL;
    LS_S4_ClipBack : BOOL;
    MachineRunStatus : BOOL;
    LS_S4_UpDownOut : BOOL;
    LS_S4_ClipOut : BOOL;
    SNR_Index : BOOL;
    RY_Index : BOOL;
    SOL_S4_THMoveOut : BOOL;
    Manual2AutoFlag : BOOL;
    HMIPB_SOL_S4_THMoveBack : BOOL;
    HMIPB_SOL_S4_THMoveOut : BOOL;
    LS_S4_THMoveOut : BOOL;
    YAMAHA_ORG : BOOL;
    SNR_S4_Feed : BOOL;
    FeedStart : ARRAY[0..19] OF BOOL;
    FeedFinish : ARRAY[0..19] OF BOOL;
    ErrorStatus_TH : ARRAY[0..19] OF BOOL;
    LS_S2_UpDownOut : BOOL;
END_VAR
(*************************************************************************
程序名稱:第4站轉子組流程
作者:蔡相偉
版本,日期,版本資訊:
1.0.0		2017/11/22		初始版本

PowerOn=0
Idle=1
上下出=2
夾取出=3
上下回=4
移位出=5
上下出=6
夾取回=7
上下回=8
移位回=9
*************************************************************************)
(*************************************************************************
異常碼
急停=1
氣缸=2
轉子組放入失敗=3
*************************************************************************)
//*************************************************************************
//本站狀態判斷
IF IndexData[4].OKFlag[4]
	OR IndexData[4].NGFlag[4] THEN
	IndexData[4].FinishFlag[4]:=TRUE;
END_IF;
IF  	IndexData[4].NGFlag[2] THEN
	IndexData[4].NGFlag[4]:=TRUE;
END_IF;

IF DisablePB[4] AND IndexData[4].FinishFlag[2] AND IndexData[4].OKFlag[2] AND NOT(IndexData[4].NGFlag[2]) THEN
	IndexData[4].OKFlag[4]:=TRUE;
END_IF;

Rtrig_test(CLK:=TestPB[4]);
//PowerOn=0
IF NOT(SystemReadyStatus AND AutoStatus AND NOT(ErrorStatus[4]) AND NOT(Error_PB_EStop)) THEN
	Autoflow:=0;
END_IF;
	//EStop異常碼
	IF Error_PB_Estop AND NOT(IndexData[4].FinishFlag[4]) AND IndexData[4].OkFlag[1] THEN
		IndexData[4].NGFlag[4]:=TRUE;
		IndexData[4].ErrorLog[4]:=1;
	END_IF;
	//Error異常碼
	IF ErrorStatus[4] AND NOT(IndexData[4].FinishFlag[4]) AND IndexData[4].OkFlag[1] THEN
		IndexData[4].NGFlag[4]:=TRUE;
		IndexData[4].ErrorLog[4]:=2;
	END_IF;
//Idle=1
IF AutoFlow=0 AND SystemReadyStatus AND AutoStatus AND NOT(ErrorStatus[4]) AND NOT(Error_PB_EStop) THEN
	AutoFlow:=1;
END_IF;

IF Autoflow=9 AND LS_S4_MoveBack THEN
	Autoflow:=1;
END_IF;

//上下出=2
IF Autoflow=1
	AND AutoStatus
	AND NOT(DisablePB[4])
	AND LS_S4_THMoveBack
	AND LS_S4_MoveBack
	AND LS_S4_UpDownBack
	AND LS_S4_ClipBack
	AND (MachineRunStatus AND NOT(IndexData[4].FinishFlag[4]) AND IndexData[4].FinishFlag[2] AND IndexData[4].OKFlag[2] AND NOT(IndexData[4].NGFlag[2])
	OR Rtrig_test.Q) THEN
	Autoflow:=2;
END_IF;

//夾取出=3
IF Autoflow=2 AND LS_S4_UpDownOut THEN
	Autoflow:=3;
END_IF;

//上下回=4
IF Autoflow=3 AND LS_S4_ClipOut THEN
	Autoflow:=4;
END_IF;

//移位出=5
IF Autoflow=4 AND LS_S4_UpDownBack THEN
	Autoflow:=5;
END_IF;

//上下出=6
IF Autoflow=5 AND LS_S4_MoveOut THEN
	Autoflow:=6;
END_IF;
TON1(In:=Autoflow=6 AND LS_S4_UpDownOut, PT:=t#500ms);		//OK
TON2(In:=Autoflow=6 AND NOT(LS_S4_UpDownOut), PT:=t#2000ms);		//NG

//夾取回=7
IF Autoflow=6 AND TON1.Q THEN
	IndexData[4].OKFlag[4]:=TRUE;
	IndexData[4].NGFlag[4]:=FALSE;
	Autoflow:=7;
END_IF;
IF Autoflow=6 AND TON2.Q THEN
	IndexData[4].OKFlag[4]:=FALSE;
	IndexData[4].NGFlag[4]:=TRUE;
	IndexData[4].ErrorLog[4]:=3;
	Autoflow:=7;
END_IF;

//上下回=8
IF Autoflow=7 AND LS_S4_ClipBack THEN
	Autoflow:=8;
END_IF;

//移位回=9
IF Autoflow=8 AND LS_S4_UpDownBack THEN
	Autoflow:=9;
END_IF;
//*************************************************************************
//手動
//移位歸電磁閥
interlockback[0]:=LS_S4_UpDownBack AND NOT(SOL_S4_UpDown);
IF ((HMIPB_SOL_S4_MoveBack AND NOT(AutoStatus)) OR Autoflow=9 OR Initflow=9) AND interlockback[0] THEN
	SOL_S4_MoveBack:=TRUE;
	SOL_S4_MoveOut:=FALSE;
END_IF;
IF LS_S4_MoveBack THEN
	SOL_S4_MoveBack:=FALSE;
END_IF;

//移位出電磁閥
interlockout[0]:=LS_S4_UpDownBack AND NOT(SOL_S4_UpDown);
IF ((HMIPB_SOL_S4_MoveOut AND NOT(AutoStatus)) OR Autoflow=5) AND interlockout[0] THEN
	SOL_S4_MoveBack:=FALSE;
	SOL_S4_MoveOut:=TRUE;
END_IF;
IF LS_S4_MoveOut THEN
	SOL_S4_MoveOut:=FALSE;
END_IF;

//上下電磁閥
R_TRIG_1[1](CLK:=HMIPB_SOL_S4_UpDown AND NOT(AutoStatus));
interlockback[1]:=TRUE;
interlockout[1]:=((LS_S4_MoveBack AND LS_S4_THMoveBack AND NOT(SOL_S4_THMoveBack) AND NOT(SOL_S4_THMoveOut)) OR
	(LS_S4_MoveOut AND SNR_Index AND NOT(RY_Index))) AND
	NOT(SOL_S4_MoveBack) AND NOT(SOL_S4_MoveOut);
(*SET*)
IF ((R_TRIG_1[1].Q AND NOT(solstatus[1])) OR Autoflow=2 OR Autoflow=6) AND interlockout[1] THEN
	SOL_S4_UpDown:=TRUE;
END_IF;
(*RESET*)
IF ((R_TRIG_1[1].Q AND (solstatus[1])) OR Autoflow=4 OR Autoflow=8 OR Initflow=8) AND interlockback[1] THEN
	SOL_S4_UpDown:=FALSE;
END_IF;
(*STATUS*)
solstatus[1]:=SOL_S4_UpDown;

//夾持電磁閥
R_TRIG_1[2](CLK:=HMIPB_SOL_S4_Clip AND NOT(AutoStatus));
interlockback[2]:=TRUE;
interlockout[2]:=TRUE;
(*SET*)
IF ((R_TRIG_1[2].Q AND NOT(solstatus[2])) OR Autoflow=3) AND interlockout[2] THEN
	SOL_S4_Clip:=TRUE;
END_IF;
(*RESET*)
IF ((R_TRIG_1[2].Q AND (solstatus[2])) OR Autoflow=7 OR Initflow=7) AND interlockback[2] THEN
	SOL_S4_Clip:=FALSE;
END_IF;
(*STATUS*)
solstatus[2]:=SOL_S4_Clip;
(*************************************************************************
程序名稱:第4站轉子組RESET流程
作者:蔡相偉
版本,日期,版本資訊:
1.0.0		2017/11/22		初始版本

PowerOn=0
Idle=1
夾取回=7
上下回=8
移位回=9
*************************************************************************)
//PowerOn=0
IF NOT(SystemReadyStatus) THEN
	Initflow:=0;
END_IF;

//Idle=1
IF Initflow=0 AND SystemReadyStatus THEN
	Initflow:=1;
END_IF;

IF Initflow=9 AND LS_S4_MoveBack THEN
	Initflow:=1;
END_IF;

//夾取回=7
F_TRIG_1(CLK:= ErrorStatus[4] OR Error_PB_Estop);
IF Initflow=1 AND (F_TRIG_1.Q OR Manual2AutoFlag) THEN
	Initflow:=7;
END_IF;

//上下回=8
IF Initflow=7 AND LS_S4_ClipBack THEN
	Initflow:=8;
END_IF;

//移位回=9
IF Initflow=8 AND LS_S4_UpDownBack THEN
	Initflow:=9;
END_IF;
END_PROGRAM

PROGRAM prStation4_TH
VAR
    interlockback : ARRAY[0..1] OF BOOL;
    interlockout : ARRAY[0..1] OF BOOL;
    Autoflow : INT;
    Initflow : INT;
    TON1 : TON;
    TON2 : TON;
    TON3 : TON;
END_VAR
VAR_EXTERNAL
    LS_S4_UpDownBack : BOOL;
    SOL_S4_UpDown : BOOL;
    LS_S4_MoveBack : BOOL;
    YAMAHA_ORG : BOOL;
    HMIPB_SOL_S4_THMoveBack : BOOL;
    AutoStatus : BOOL;
    SOL_S4_THMoveBack : BOOL;
    SOL_S4_THMoveOut : BOOL;
    LS_S4_THMoveBack : BOOL;
    HMIPB_SOL_S4_THMoveOut : BOOL;
    LS_S4_THMoveOut : BOOL;
    SystemReadyStatus : BOOL;
    ErrorStatus : ARRAY[0..19] OF BOOL;
    Error_PB_EStop : BOOL;
    IndexData : ARRAY[0..19] OF stIndexData;
    ErrorStatus_TH : ARRAY[0..19] OF BOOL;
    SNR_S4_Feed : BOOL;
    FeedStart : ARRAY[0..19] OF BOOL;
    FeedFinish : ARRAY[0..19] OF BOOL;
    Error_SNR_S4_Feed : BOOL;
    PB_Reset : BOOL;
END_VAR
(*************************************************************************
程序名稱:第4站轉子組節流流程
作者:蔡相偉
版本,日期,版本資訊:
1.0.0		2017/11/22		初始版本

PowerOn=0
Idle=1
無料節流出=2
送料開始=3
送料中=4
送料完成=5
節流回=6
檢查有無料=7
*************************************************************************)
//PowerOn=0
IF NOT(SystemReadyStatus AND AutoStatus AND NOT(ErrorStatus_TH[4]) AND NOT(Error_PB_EStop)) THEN
	Autoflow:=0;
END_IF;

//Idle=1
IF AutoFlow=0 AND SystemReadyStatus AND AutoStatus AND NOT(ErrorStatus[4]) AND NOT(Error_PB_EStop) THEN
	AutoFlow:=1;
END_IF;

IF Autoflow=7 AND (TON2.Q OR TON3.Q) THEN
	Autoflow:=1;
END_IF;

//無料節流出=2
TON1(In:=Autoflow=1 AND NOT(SNR_S4_Feed), PT:=t#1s);
IF AutoFlow=1 AND TON1.Q AND NOT(Error_SNR_S4_Feed) THEN
	AutoFlow:=2;
END_IF;

//送料開始=3
IF Autoflow=2 AND LS_S4_THMoveOut THEN
	Autoflow:=3;
END_IF;
IF Autoflow=3 THEN
	FeedStart[4]:=TRUE;
END_IF;
IF FeedFinish[4] THEN
	FeedStart[4]:=FALSE;
END_IF;

//送料中=4
IF Autoflow=3 AND FeedStart[4] THEN
	Autoflow:=4;
END_IF;

//送料完成=5
IF Autoflow=4 AND NOT(FeedStart[4]) THEN
	Autoflow:=5;
END_IF;

//節流回=6
IF Autoflow=5 THEN
	Autoflow:=6;
END_IF;

//檢查有無料=7
IF Autoflow=6 AND LS_S4_THMoveBack THEN
	Autoflow:=7;
END_IF;
TON2(In:=Autoflow=7 AND (SNR_S4_Feed), PT:=t#300ms); 			//OK
TON3(In:=Autoflow=7 AND NOT(SNR_S4_Feed), PT:=t#300ms);	//NG
IF TON3.Q THEN
	Error_SNR_S4_Feed:=TRUE;
END_IF;
IF PB_Reset THEN
	Error_SNR_S4_Feed:=FALSE;
END_IF;

//*************************************************************************
//手動
//節流移位歸電磁閥
interlockback[0]:=((LS_S4_UpDownBack AND NOT(SOL_S4_UpDown)) OR NOT(LS_S4_MoveBack)) AND YAMAHA_ORG;
IF ((HMIPB_SOL_S4_THMoveBack AND NOT(AutoStatus)) OR Autoflow=6 OR ErrorStatus_TH[4]) AND interlockback[0] THEN
	SOL_S4_THMoveBack:=TRUE;
	SOL_S4_THMoveOut:=FALSE;
END_IF;
IF LS_S4_THMoveBack THEN
	SOL_S4_THMoveBack:=FALSE;
END_IF;

//節流移位出電磁閥
interlockout[0]:=((LS_S4_UpDownBack AND NOT(SOL_S4_UpDown)) OR NOT(LS_S4_MoveBack)) AND YAMAHA_ORG;
IF ((HMIPB_SOL_S4_THMoveOut AND NOT(AutoStatus)) OR Autoflow=2) AND interlockout[0] THEN
	SOL_S4_THMoveBack:=FALSE;
	SOL_S4_THMoveOut:=TRUE;
END_IF;
IF LS_S4_THMoveOut THEN
	SOL_S4_THMoveOut:=FALSE;
END_IF;
END_PROGRAM

PROGRAM prStation2
VAR
    interlockback : ARRAY[0..1] OF BOOL;
    interlockout : ARRAY[0..1] OF BOOL;
    solstatus : ARRAY[0..1] OF BOOL;
    R_TRIG_1 : ARRAY[0..1] OF R_TRIG;
    Rtrig_test : R_TRIG;
    F_TRIG_1 : F_TRIG;
    Autoflow : INT;
    Initflow : INT;
    TON1 : TON;
    TON2 : TON;
END_VAR
VAR_EXTERNAL
    IndexData : ARRAY[0..19] OF stIndexData;
    DisablePB : ARRAY[0..19] OF BOOL;
    SystemReadyStatus : BOOL;
    AutoStatus : BOOL;
    ErrorStatus : ARRAY[0..19] OF BOOL;
    Error_PB_EStop : BOOL;
    LS_S2_UpDownBack : BOOL;
    MachineRunStatus : BOOL;
    LS_S2_UpDownOut : BOOL;
    HMIPB_SOL_S2_UpDown : BOOL;
    SNR_Index : BOOL;
    RY_Index : BOOL;
    SOL_S2_UpDown : BOOL;
    Manual2AutoFlag : BOOL;
    TestPB : ARRAY[0..19] OF BOOL;
END_VAR
(*************************************************************************
程序名稱:第2站檢查下夾板流程
作者:蔡相偉
版本,日期,版本資訊:
1.0.0		2017/11/22		初始版本

